// ---- POUs/Station/FB_StationTakeLoad.TcPOU
FUNCTION_BLOCK FB_StationTakeLoad
VAR_INPUT
	Enable:				BOOL;
	System:				REFERENCE TO ST_System;
	Station:			REFERENCE TO ST_SystemStation;
	Error:				REFERENCE TO ST_Error;
	Setting:			REFERENCE TO ST_Setting;
	Recipe:				REFERENCE TO ST_Recipe;	
	Parameter:			REFERENCE TO ST_StationTakeLoad;
END_VAR
VAR_OUTPUT
END_VAR
VAR
	_i:					INT;
	_arrTon:		    ARRAY[0..20] OF TON;
	_arrFbErrorTag:		ARRAY[0..20] OF FB_ErrorTag;
	_arrState:			ARRAY[0..20] OF BOOL;
	
	_iMoveAbsIndex1:	UINT;
	_iMoveAbsIndex2:	UINT;
	_bIsZWork:			BOOL;// 取Line0为真 其他情况为假
	_stHandshake: ST_StationTakeLoadHandshake;
END_VAR

A_Auto();
A_Home();

ACTION A_Auto:
CASE Station.iStepNow OF
	1000:
		Station.arrInfo[E_Language.Chinese]:="初始化完成 等待启动";
		IF Enable THEN
			Station.iStepNext:=1101;
		END_IF
	1101:
		Station.arrInfo[E_Language.Chinese]:="取料信号判断";
		Parameter.eState:=E_StationState.Load;
		Setting.eTakeModeBuffer:=E_TakeMode.None;
		Station.iStepNext:=1111;
	1111:
		IF Setting.eTakeModeBuffer=E_TakeMode.None THEN
			Setting.eTakeModeBuffer:=Setting.eTakeMode;
		ELSE
			Parameter.eState:=E_StationState.Busy;
			Station.iStepNext:=1151;
		END_IF
	1151:
		Station.arrInfo[E_Language.Chinese]:="请求取料";
		CASE Setting.eTakeModeBuffer OF
			E_TakeMode.Take0:
				_iMoveAbsIndex1:=2;
				_bIsZWork:=TRUE;
				Parameter.stHandshake.bRequestLine0Buffer_T0 :=TRUE;
				IF Parameter.stHandshake.bResponseTake_T0 THEN
					Station.iStepNext:=1201;
				END_IF
			E_TakeMode.Take1:
				_iMoveAbsIndex1:=3;
				_bIsZWork:=FALSE;
				Parameter.stHandshake.bRequestLineLoad_T1:=TRUE;
				IF Parameter.stHandshake.bResponseTake_T1 THEN
					Station.iStepNext:=1201;
				END_IF
			E_TakeMode.Take3Load:
				_iMoveAbsIndex1:=4;
				_bIsZWork:=FALSE;
				Parameter.stHandshake.bRequestLineLoad_T3:=TRUE;
				IF Parameter.stHandshake.bResponseTake_T3 THEN
					Station.iStepNext:=1201;
				END_IF
			E_TakeMode.None:
				Station.iStepNext:=1101;
		END_CASE
	1201:
		Station.arrInfo[E_Language.Chinese]:="Y轴至取料位";
		Parameter.eState:=E_StationState.Busy;
		IF Parameter.fbTakeY.M_MoveAbs(_iMoveAbsIndex1) THEN
			Station.iStepNext:=1301;
		END_IF
	1301:
		Station.arrInfo[E_Language.Chinese]:="Z模组下降";
		IF M_ZWork()  THEN
			Station.iStepNext:=1401;
		END_IF
	1401:
		Station.arrInfo[E_Language.Chinese]:="夹紧气缸夹紧";
		IF Parameter.fbTakeClamp.M_WorkRequest() THEN
			Station.iStepNext:=1501;
		END_IF
	1501:
		Station.arrInfo[E_Language.Chinese]:="Z模组上升";
		IF M_ZHome() THEN
			Station.iStepNext:=1511;
		END_IF
	1511:
		Station.arrInfo[E_Language.Chinese]:="复位取料请求 ";
		CASE Setting.eTakeModeBuffer OF
			E_TakeMode.Take0:
				Parameter.stHandshake.bRequestLine0Buffer_T0 :=FALSE;
				IF NOT Parameter.stHandshake.bResponseTake_T0 THEN
					Station.iStepNext:=1601;
				END_IF
			E_TakeMode.Take1:
				Parameter.stHandshake.bRequestLineLoad_T1:=FALSE;
				IF NOT Parameter.stHandshake.bResponseTake_T1 THEN
					Station.iStepNext:=1601;
				END_IF
			E_TakeMode.Take3Load:
				Parameter.stHandshake.bRequestLineLoad_T3:=FALSE;
				IF NOT Parameter.stHandshake.bResponseTake_T3 THEN
					Station.iStepNext:=1601;
				END_IF
		END_CASE
	1601:
		Station.arrInfo[E_Language.Chinese]:="请求放料";
		Parameter.eState:=E_StationState.Done;
		Setting.eTakeModeBuffer:=E_TakeMode.None;
		Station.iStepNext:=1611;
	1611:
		IF Setting.eTakeModeBuffer=E_TakeMode.None THEN
			Setting.eTakeModeBuffer:=Setting.eTakeMode;
		ELSE
			Parameter.eState:=E_StationState.Busy;
			Station.iStepNext:=1651;
		END_IF
	1651:
		_bIsZWork:=FALSE;
		CASE Setting.eTakeModeBuffer OF
			E_TakeMode.Place1:
				_iMoveAbsIndex2:=3;
				Parameter.stHandshake.bRequestLineLoad_P1:=TRUE;
				IF Parameter.stHandshake.bResponseTake_P1 THEN
					Station.iStepNext:=1701;
				END_IF
			E_TakeMode.Place3Load:
				_iMoveAbsIndex2:=4;
				Parameter.stHandshake.bRequestLineLoad_P3:=TRUE;
				IF Parameter.stHandshake.bResponseTake_P3 THEN
					Station.iStepNext:=1701;
				END_IF
		END_CASE
	1701:
		Station.arrInfo[E_Language.Chinese]:="等待Y轴至放料位";
		IF Parameter.fbTakeY.M_MoveAbs(_iMoveAbsIndex2) THEN
			Station.iStepNext:=1801;
		END_IF
	1801:
		Station.arrInfo[E_Language.Chinese]:="Z模组下降";
		IF M_ZWork() THEN
			Station.iStepNext:=1901;
		END_IF
	1901:
		Station.arrInfo[E_Language.Chinese]:="夹紧气缸松开";
		IF Parameter.fbTakeClamp.M_HomeRequest() THEN
			Station.iStepNext:=2001;
		END_IF
	2001:
		Station.arrInfo[E_Language.Chinese]:="Z模组上升";
		IF M_ZHome() THEN
			Station.iStepNext:=2101;
		END_IF
	2101:
		Station.arrInfo[E_Language.Chinese]:="复位放料请求";
		CASE Setting.eTakeModeBuffer OF
			E_TakeMode.Place1:
				Parameter.stHandshake.bRequestLineLoad_P1:=FALSE;
				IF NOT Parameter.stHandshake.bResponseTake_P1 THEN
					Station.iStepNext:=2201;
				END_IF
			E_TakeMode.Place3Load:
				Parameter.stHandshake.bRequestLineLoad_P3:=FALSE;
				IF NOT Parameter.stHandshake.bResponseTake_P3 THEN
					Station.iStepNext:=2201;
				END_IF
		END_CASE
	2201:
		Station.arrInfo[E_Language.Chinese]:="Y轴至初始位";
		IF Parameter.fbTakeY.M_MoveAbs(1) THEN
			Station.iStepNext:=1101;
		END_IF
END_CASE
END_ACTION

ACTION A_Home:
CASE Station.iStepNow OF
	0:
		Station.arrInfo[E_Language.Chinese]:="等待初始化";
		Parameter.stHandshake:=_stHandshake;
		Parameter.eState:=E_StationState.None;
		Setting.eTakeModeBuffer:=E_TakeMode.None;
		Station.iStepNext:=SEL(Enable,1000,500);
	500:
		Station.arrInfo[E_Language.Chinese]:="夹紧气缸松开";
		IF Parameter.fbTakeClamp.M_HomeRequest() THEN
			Station.iStepNext:=600;
		END_IF
	600:
		Station.arrInfo[E_Language.Chinese]:="Z模组初始化";
		IF M_ZInit() THEN
			Station.iStepNext:=700;
		END_IF
	700:
		Station.arrInfo[E_Language.Chinese]:="Z模组至上升位";
		IF M_ZHome() THEN
			Station.iStepNext:=800;
		END_IF
	800:
		Station.arrInfo[E_Language.Chinese]:="Y模组回零";
		IF Parameter.fbTakeY.M_Home() THEN
			Station.iStepNext:=900;
		END_IF
	900:
		Station.arrInfo[E_Language.Chinese]:="Y模组至初始位";
		IF Parameter.fbTakeY.M_MoveAbs(1) THEN
			Station.iStepNext:=1000;
		END_IF
END_CASE
END_ACTION

METHOD M_ZHome : BOOL
VAR_INPUT
END_VAR
CASE Recipe.eMachineType OF
	E_MachineType.LH311,E_MachineType.RH311:
		M_ZHome:=Parameter.fbTakeLift1.M_HomeRequest() AND Parameter.fbTakeLift2.M_HomeRequest();
	E_MachineType.LH353,E_MachineType.RH353:
		M_ZHome:=Parameter.fbTakeZ.M_MoveAbs(1);
	E_MachineType.LH367,E_MachineType.RH367:
		M_ZHome:=Parameter.fbTakeLift1.M_HomeRequest() AND Parameter.fbTakeLift2.M_HomeRequest();
	E_MachineType.LH201,E_MachineType.RH201:
		M_ZHome:=Parameter.fbTakeZ.M_MoveAbs(1);
	E_MachineType.LH069,E_MachineType.RH069:
		M_ZHome:=Parameter.fbTakeZ.M_MoveAbs(1);
	E_MachineType.LH373,E_MachineType.RH373:
		M_ZHome:=Parameter.fbTakeZ.M_MoveAbs(1);
END_CASE
END_METHOD

METHOD M_ZInit : BOOL
VAR_INPUT
END_VAR
CASE Recipe.eMachineType OF
	E_MachineType.LH311,E_MachineType.RH311:
		M_ZInit:=TRUE;
	E_MachineType.LH353,E_MachineType.RH353:
		M_ZInit:=Parameter.fbTakeZ.M_Home();
	E_MachineType.LH367,E_MachineType.RH367:
		M_ZInit:=TRUE;
	E_MachineType.LH201,E_MachineType.RH201:
		M_ZInit:=Parameter.fbTakeZ.M_Home();
	E_MachineType.LH069,E_MachineType.RH069:
		M_ZInit:=Parameter.fbTakeZ.M_Home();
	E_MachineType.LH373,E_MachineType.RH373:
		M_ZInit:=Parameter.fbTakeZ.M_Home();
END_CASE
END_METHOD

METHOD M_ZWork : BOOL
VAR_INPUT
END_VAR
CASE Recipe.eMachineType OF
	E_MachineType.LH311,E_MachineType.RH311:
		M_ZWork:=Parameter.fbTakeLift1.M_WorkRequest() AND Parameter.fbTakeLift2.M_WorkRequest();
	E_MachineType.LH353,E_MachineType.RH353:
		M_ZWork:=SEL(_bIsZWork,Parameter.fbTakeZ.M_MoveAbs(3) ,Parameter.fbTakeZ.M_MoveAbs(2));
	E_MachineType.LH367,E_MachineType.RH367:
		M_ZWork:=Parameter.fbTakeLift1.M_WorkRequest() AND SEL(_bIsZWork,TRUE ,Parameter.fbTakeLift2.M_WorkRequest()) ;
	E_MachineType.LH201,E_MachineType.RH201:
		M_ZWork:=SEL(_bIsZWork,Parameter.fbTakeZ.M_MoveAbs(3) ,Parameter.fbTakeZ.M_MoveAbs(2));
	E_MachineType.LH069,E_MachineType.RH069:
		M_ZWork:=SEL(_bIsZWork,Parameter.fbTakeZ.M_MoveAbs(3) ,Parameter.fbTakeZ.M_MoveAbs(2));
	E_MachineType.LH373,E_MachineType.RH373:
		M_ZWork:=SEL(_bIsZWork,Parameter.fbTakeZ.M_MoveAbs(3) ,Parameter.fbTakeZ.M_MoveAbs(2));
END_CASE
END_METHOD

END_FUNCTION_BLOCK

// ---- POUs/Station/FB_StationDismantling.TcPOU
FUNCTION_BLOCK FB_StationDismantling
VAR_INPUT
	Enable:				BOOL;
	System:				REFERENCE TO ST_System;
	Station:			REFERENCE TO ST_SystemStation;
	Error:				REFERENCE TO ST_Error;
	Setting:			REFERENCE TO ST_Setting;
	Recipe:				REFERENCE TO ST_Recipe;	
	Parameter:			REFERENCE TO ST_StationDismantling;	
END_VAR
VAR_OUTPUT
END_VAR
VAR
	_i:					INT;
	_arrTon:		    ARRAY[0..20] OF TON;
	_arrFbErrorTag:		ARRAY[0..20] OF FB_ErrorTag;
	_arrState:			ARRAY[0..20] OF BOOL;
	_bOpenLockTemp:		BOOL;
	_bResetLockTemp:	BOOL;
	_stHandshake:		ST_StationDismantlingHandshake;
END_VAR

A_Home();
A_Auto();

ACTION A_Auto:
CASE Station.iStepNow OF
	1000:
		Station.arrInfo[E_Language.Chinese]:="初始化完成 等待启动";
		IF  Enable THEN
			Station.iStepNext:=1101;
		END_IF
	1101:
		Station.arrInfo[E_Language.Chinese]:="判断是否有料";
		Parameter.eState:=E_StationState.Busy;
		IF NOT Parameter.bClose AND NOT Parameter.bPalletCheck2 THEN
			Station.iStepNext:=1201;
		END_IF
	1201:
		Station.arrInfo[E_Language.Chinese]:="请求放料";
		Parameter.eState:=E_StationState.Load;
		Station.iStepNext:=1301;
	1301:
		Parameter.stHandshake.bRequestLineLoad_D:=TRUE;
		IF Parameter.stHandshake.bResponseDismantling_D THEN
			Parameter.eState:=E_StationState.Busy;
			Station.iStepNext:=1401;
		END_IF
	1401:
		Station.arrInfo[E_Language.Chinese]:="等待产品流入";
		IF Parameter.bPalletCheck2 THEN
			Station.iStepNext:=1501;
		END_IF
	1501:
		Station.arrInfo[E_Language.Chinese]:="复位放料请求";
		Parameter.stHandshake.bRequestLineLoad_D:=FALSE;
		IF NOT Parameter.stHandshake.bResponseDismantling_D THEN
			Station.iStepNext:=1601;
		END_IF
	1601:
		Station.arrInfo[E_Language.Chinese]:="等待产品到位";
		IF Parameter.bPalletCheck2 THEN
			Station.iStepNext:=1701;
		END_IF
	1701:
		Station.arrInfo[E_Language.Chinese]:="顶升气缸上升 阻挡气缸缩回";
		_bOpenLockTemp:=FALSE;
		_arrState[0]:=Parameter.fbLift.M_WorkRequest() ;
		_arrState[1]:=Parameter.fbPrevent.M_HomeRequest();
		IF _arrState[0] AND _arrState[1]THEN
			Station.iStepNext:=1801;
		END_IF
	1801:
		Station.arrInfo[E_Language.Chinese]:="载具解锁";
		IF M_OpenLock() THEN
			Station.iStepNext:=1901;
		END_IF
	1901:
		Station.arrInfo[E_Language.Chinese]:="校平气缸伸出";
		IF M_StandardWork() THEN
			Station.iStepNext:=2001;
		END_IF
	2001:
		Station.arrInfo[E_Language.Chinese]:="请求取UC";
		Parameter.stHandshake.bRequestUc:=TRUE;
		IF Parameter.stHandshake.bResponseDismantling_Uc THEN
			Station.iStepNext:=2201;
		END_IF
	2201:
		Parameter.stHandshake.bRequestUc:=FALSE;
		IF NOT Parameter.stHandshake.bResponseDismantling_Uc THEN
			Station.iStepNext:=2301;
		END_IF
	2301:
		Station.arrInfo[E_Language.Chinese]:="校平气缸缩回";
		_bResetLockTemp:=FALSE;
		IF M_StandardHome() THEN
			Station.iStepNext:=2401;
		END_IF
	2401:
		Station.arrInfo[E_Language.Chinese]:="载具复位";
		IF M_ResetLock() THEN
			Station.iStepNext:=2501;
		END_IF
	2501:
		Station.arrInfo[E_Language.Chinese]:="判断下工装站是否屏蔽";
		IF NOT  Parameter.bCloseUnloadElevator THEN
			Station.iStepNext:=2551;
		ELSIF Parameter.fbLift.M_HomeRequest() THEN
			Station.iStepNext:=2801;
		END_IF
	2551:
		Station.arrInfo[E_Language.Chinese]:="请求下工装";
		Parameter.stHandshake.bRequestElevator:=TRUE;
		IF Parameter.stHandshake.bResponseDismantling_E THEN
			Station.iStepNext:=2601;
		END_IF
	2601:
		Station.arrInfo[E_Language.Chinese]:="顶升气缸下降";
		IF Parameter.fbLift.M_HomeRequest() THEN
			Station.iStepNext:=2701;
		END_IF
	2701:
		Station.arrInfo[E_Language.Chinese]:="复位请求";
		Parameter.stHandshake.bRequestElevator:=FALSE;
		IF NOT Parameter.stHandshake.bResponseDismantling_E THEN
			Station.iStepNext:=2801;
		END_IF
	2801:
		Station.arrInfo[E_Language.Chinese]:="等待产品流出";
		IF NOT Parameter.bPalletCheck1 AND NOT Parameter.bPalletCheck2 AND NOT Parameter.bPalletCheck3 THEN
			Station.iStepNext:=2901;
		END_IF
	2901:
		Station.arrInfo[E_Language.Chinese]:="阻挡气缸伸出";
		IF  Parameter.fbPrevent.M_WorkRequest() THEN
			Station.iStepNext:=1101;
		END_IF
END_CASE
END_ACTION

ACTION A_Home:
CASE Station.iStepNow OF
	0:
		Station.arrInfo[E_Language.Chinese]:="等待初始化";
		Parameter.stHandshake:=_stHandshake;
		Parameter.eState:=E_StationState.Done;
		Station.iStepNext:=SEL(Enable,1000,100);
	100:
		Station.arrInfo[E_Language.Chinese]:="阻挡气缸伸出";
		IF Parameter.fbPrevent.M_WorkRequest() THEN
			Station.iStepNext:=200;
		END_IF
	200:
		Station.arrInfo[E_Language.Chinese]:="侧推气缸缩回";
		IF M_LateralHome() THEN
			Station.iStepNext:=300;
		END_IF
	300:
		Station.arrInfo[E_Language.Chinese]:="旋转气缸复位";
		IF Parameter.fbRotate.M_HomeRequest() THEN
			Station.iStepNext:=400;
		END_IF
	400:
		Station.arrInfo[E_Language.Chinese]:="校平气缸缩回";
		IF M_StandardHome() THEN
			Station.iStepNext:=500;
		END_IF
	500:
		Station.arrInfo[E_Language.Chinese]:="顶升气缸缩回";
		IF Parameter.fbLift.M_HomeRequest() THEN
			Station.iStepNext:=1000;
		END_IF
END_CASE
END_ACTION

METHOD M_LateralHome : BOOL
VAR_INPUT
END_VAR
VAR
	_temp:			ARRAY[0..10] OF BOOL;
END_VAR
CASE Recipe.eMachineType OF
	E_MachineType.LH311,E_MachineType.RH311:
		M_LateralHome:=Parameter.fbLateral1.M_HomeRequest();
	E_MachineType.LH353,E_MachineType.RH353:
		_temp[0]:=Parameter.fbLateral1.M_HomeRequest();
		_temp[1]:=Parameter.fbLateral2.M_HomeRequest();
		M_LateralHome:=_temp[0] AND _temp[1];
	E_MachineType.LH367,E_MachineType.RH367:
		_temp[0]:=Parameter.fbLateral1.M_HomeRequest();
		_temp[1]:=Parameter.fbLateral2.M_HomeRequest();
		M_LateralHome:=_temp[0] AND _temp[1];
	E_MachineType.LH201,E_MachineType.RH201:
		_temp[0]:=Parameter.fbLateral1.M_HomeRequest();
		_temp[1]:=Parameter.fbLateral2.M_HomeRequest();
		M_LateralHome:=_temp[0] AND _temp[1];
	E_MachineType.LH069,E_MachineType.RH069:
		_temp[0]:=Parameter.fbLateral1.M_HomeRequest();
		_temp[1]:=Parameter.fbLateral2.M_HomeRequest();
		M_LateralHome:=_temp[0] AND _temp[1];
	E_MachineType.LH373,E_MachineType.RH373:
		M_LateralHome:=Parameter.fbLateral1.M_HomeRequest();
END_CASE
END_METHOD

METHOD M_LateralWork : BOOL
VAR_INPUT
END_VAR

VAR
	_temp: array[0..10] of bool;
END_VAR
CASE Recipe.eMachineType OF
	E_MachineType.LH311,E_MachineType.RH311:
		M_LateralWork:=Parameter.fbLateral1.M_WorkRequest();
	E_MachineType.LH353,E_MachineType.RH353:
		_temp[0]:=Parameter.fbLateral1.M_WorkRequest();
		_temp[1]:=Parameter.fbLateral2.M_WorkRequest();
		M_LateralWork:=_temp[0] AND _temp[1];
	E_MachineType.LH367,E_MachineType.RH367:
		_temp[0]:=Parameter.fbLateral1.M_WorkRequest();
		_temp[1]:=Parameter.fbLateral2.M_WorkRequest();
		M_LateralWork:=_temp[0] AND _temp[1];
	E_MachineType.LH201,E_MachineType.RH201:
		_temp[0]:=Parameter.fbLateral1.M_WorkRequest();
		_temp[1]:=Parameter.fbLateral2.M_WorkRequest();
		M_LateralWork:=_temp[0] AND _temp[1];
	E_MachineType.LH069,E_MachineType.RH069:
		_temp[0]:=Parameter.fbLateral1.M_WorkRequest();
		_temp[1]:=Parameter.fbLateral2.M_WorkRequest();
		M_LateralWork:=_temp[0] AND _temp[1];
	E_MachineType.LH373,E_MachineType.RH373:
		M_LateralWork:=Parameter.fbLateral1.M_WorkRequest();
END_CASE
END_METHOD

METHOD M_OpenLock : BOOL
VAR_INPUT
END_VAR
IF Recipe.eMachineType=E_MachineType.LH311 OR Recipe.eMachineType=E_MachineType.RH311 THEN
	IF M_LateralWork() THEN
		M_OpenLock:=Parameter.fbRotate.M_WorkRequest();
	END_IF
ELSE
	IF NOT _bOpenLockTemp THEN
		IF M_LateralWork() THEN
			_bOpenLockTemp:=Parameter.fbRotate.M_WorkRequest();
		END_IF
	ELSE
		CASE  Recipe.eMachineType OF
			E_MachineType.LH201,E_MachineType.RH201:
				M_OpenLock:=Parameter.fbLateral2.M_HomeRequest();
			ELSE
				M_OpenLock:=M_LateralHome();
		END_CASE
	END_IF
END_IF
END_METHOD

METHOD M_ResetLock : BOOL
VAR_INPUT
END_VAR
IF Recipe.eMachineType=E_MachineType.LH311 OR Recipe.eMachineType=E_MachineType.RH311 THEN
	IF M_LateralHome() THEN
		M_ResetLock:=Parameter.fbRotate.M_HomeRequest();;
	END_IF
ELSE
	IF NOT _bResetLockTemp THEN
		IF Parameter.fbLateral1.M_WorkRequest() THEN
			_bResetLockTemp:=Parameter.fbRotate.M_HomeRequest();
		END_IF
	ELSE
		M_ResetLock:=Parameter.fbLateral1.M_HomeRequest();
	END_IF
END_IF
END_METHOD

METHOD M_StandardHome : BOOL
VAR_INPUT
END_VAR
VAR
	_temp:			ARRAY[0..10] OF BOOL;
END_VAR
CASE Recipe.eMachineType OF
	E_MachineType.LH311,E_MachineType.RH311:
		_temp[0]:=Parameter.fbStandard1.M_HomeRequest();
		_temp[1]:=Parameter.fbStandard2.M_HomeRequest();
		M_StandardHome:=_temp[0] AND _temp[1];
	E_MachineType.LH353,E_MachineType.RH353:
		M_StandardHome:=Parameter.fbStandard1.M_HomeRequest();
	E_MachineType.LH367,E_MachineType.RH367:
		M_StandardHome:=Parameter.fbStandard1.M_HomeRequest();
	E_MachineType.LH201,E_MachineType.RH201:
		M_StandardHome:=TRUE;
	E_MachineType.LH069,E_MachineType.RH069:
		M_StandardHome:=TRUE;
	E_MachineType.LH373,E_MachineType.RH373:
		M_StandardHome:=Parameter.fbStandard1.M_HomeRequest();
END_CASE
END_METHOD

METHOD M_StandardWork : BOOL
VAR_INPUT
END_VAR

VAR
	_temp: array[0..10] of bool;
END_VAR
CASE Recipe.eMachineType OF
	E_MachineType.LH311,E_MachineType.RH311:
		_temp[0]:=Parameter.fbStandard1.M_WorkRequest();
		_temp[1]:=Parameter.fbStandard2.M_WorkRequest();
		M_StandardWork:=_temp[0] AND _temp[1];
	E_MachineType.LH353,E_MachineType.RH353:
		M_StandardWork:=Parameter.fbStandard1.M_WorkRequest();
	E_MachineType.LH367,E_MachineType.RH367:
		M_StandardWork:=Parameter.fbStandard1.M_WorkRequest();
	E_MachineType.LH201,E_MachineType.RH201:
		M_StandardWork:=TRUE;
	E_MachineType.LH069,E_MachineType.RH069:
		M_StandardWork:=TRUE;
	E_MachineType.LH373,E_MachineType.RH373:
		M_StandardWork:=TRUE;//Parameter.fbStandard1.M_WorkRequest();
END_CASE
END_METHOD

END_FUNCTION_BLOCK

// ---- POUs/Station/FB_StationLine0Load.TcPOU
FUNCTION_BLOCK FB_StationLine0Load
VAR_INPUT
	Enable:				BOOL;
	System:				REFERENCE TO ST_System;
	Station:			REFERENCE TO ST_SystemStation;
	Error:				REFERENCE TO ST_Error;
	Setting:			REFERENCE TO ST_Setting;
	Recipe:				REFERENCE TO ST_Recipe;	
	Parameter:			REFERENCE TO ST_StationLine0Load;
END_VAR
VAR_OUTPUT
END_VAR
VAR
	_i:					INT;
	_arrTon:		    ARRAY[0..20] OF TON;
	_arrFbErrorTag:		ARRAY[0..20] OF FB_ErrorTag;
	_arrState:			ARRAY[0..20] OF BOOL;
	
	_stHandshake:		ST_StationLine0LoadHandshake;
END_VAR

A_Home();
A_Auto();

ACTION A_Auto:
CASE Station.iStepNow OF
	1000:
		Station.arrInfo[E_Language.Chinese]:="初始化完成 等待启动";
		IF Enable THEN
			Station.iStepNext:=1100;
		END_IF
	1100:
		Station.arrInfo[E_Language.Chinese]:="判断阻挡位是否有料";
		IF Parameter.bPreventCheck THEN
			Station.iStepNext:=1601;
		ELSE
			Station.iStepNext:=1201;
		END_IF
	1201:
		Station.arrInfo[E_Language.Chinese]:="判断分料位是否有料";
		IF Parameter.bPartCheck AND Recipe.eLoadClose<>E_LoadClose.Line0 THEN
			Station.iStepNext:=1301;
		END_IF
	1301:
		Station.arrInfo[E_Language.Chinese]:="分料气缸缩回";
		IF  Parameter.fbPart.M_HomeRequest() THEN
			Station.iStepNext:=1401;
		END_IF
	1401:
		Station.arrInfo[E_Language.Chinese]:="等待产品至阻挡位";
		IF Parameter.bPreventCheck THEN
			Station.iStepNext:=1501;
		END_IF
	1501:
		Station.arrInfo[E_Language.Chinese]:="分料气缸伸出";
		IF  Parameter.fbPart.M_WorkRequest() THEN
			Station.iStepNext:=1601;
		END_IF
	1601:
		Station.arrInfo[E_Language.Chinese]:="等待缓存工站请求放料";
		IF Parameter.stHandshake.bRequestLine0Load THEN
			Parameter.stHandshake.bResponseLine0Buffer:=TRUE;
			Station.iStepNext:=1701;
		END_IF
	1701:
		Station.arrInfo[E_Language.Chinese]:="阻挡气缸缩回";
		IF Parameter.fbPrevent.M_HomeRequest() THEN
			Station.iStepNext:=1751;
		END_IF
	1751:
		Station.arrInfo[E_Language.Chinese]:="等待产品流出";
		IF NOT Parameter.bPreventCheck THEN
			Station.iStepNext:=1801;
		END_IF
	1801:
		Station.arrInfo[E_Language.Chinese]:="等待放料完成";
		IF NOT Parameter.stHandshake.bRequestLine0Load THEN
			Parameter.stHandshake.bResponseLine0Buffer:=FALSE;
			Station.iStepNext:=1901;
		END_IF
	1901:
		Station.arrInfo[E_Language.Chinese]:="阻挡气缸伸出";
		IF Parameter.fbPrevent.M_WorkRequest() THEN
			Station.iStepNext:=1100;
		END_IF
END_CASE
END_ACTION

ACTION A_Home:
CASE Station.iStepNow OF
	0:
		Station.arrInfo[E_Language.Chinese]:="等待初始化";
		Parameter.stHandshake:=_stHandshake;
		Station.iStepNext:=SEL(Enable,1000,200);
	200:
		Station.arrInfo[E_Language.Chinese]:="分料气缸 阻挡气缸伸出";
		_arrState[0]:=Parameter.fbPart.M_WorkRequest();
		_arrState[1]:=Parameter.fbPrevent.M_WorkRequest();
		IF _arrState[0] AND _arrState[1] THEN
			Station.iStepNext:=1000;
		END_IF
END_CASE
END_ACTION

END_FUNCTION_BLOCK

// ---- POUs/Station/FB_StationLine0Buffer.TcPOU
FUNCTION_BLOCK FB_StationLine0Buffer
VAR_INPUT
	Enable:				BOOL;
	System:				REFERENCE TO ST_System;
	Station:			REFERENCE TO ST_SystemStation;
	Error:				REFERENCE TO ST_Error;
	Setting:			REFERENCE TO ST_Setting;
	Recipe:				REFERENCE TO ST_Recipe;	
	Parameter:			REFERENCE TO ST_StationLine0Buffer;	
END_VAR
VAR_OUTPUT
END_VAR
VAR
	_i:					INT;
	_arrTon:		    ARRAY[0..20] OF TON;
	_arrFbErrorTag:		ARRAY[0..20] OF FB_ErrorTag;
	_arrState:			ARRAY[0..20] OF BOOL;
	
	_stHandshake:		ST_StationLine0BufferHandshake;
END_VAR

A_Home();
A_Auto();

ACTION A_Auto:
CASE Station.iStepNow OF
	1000:
		Station.arrInfo[E_Language.Chinese]:="初始化完成 等待启动";
		IF Enable THEN
			Station.iStepNext:=1101;
		END_IF
	1101:
		Station.arrInfo[E_Language.Chinese]:="判断缓存位是否有料";
		Parameter.eState:=E_StationState.Busy;
		IF Parameter.bPlace AND NOT GVL.stSetting.bDryRun THEN
			Station.iStepNext:=1501;
		ELSE
			Station.iStepNext:=1201;
		END_IF
	1201:
		Station.arrInfo[E_Language.Chinese]:="请求上料站放料";
		Parameter.stHandshake.bRequestLine0Load:=TRUE;
		IF Parameter.stHandshake.bResponseLine0Buffer THEN
			Station.iStepNext:=1301;
		END_IF
	1301:
		Station.arrInfo[E_Language.Chinese]:="等待产品到位";
		IF Parameter.bPlace THEN
			Station.iStepNext:=1401;
		END_IF
	1401:
		Station.arrInfo[E_Language.Chinese]:="复位请求信号";
		Parameter.stHandshake.bRequestLine0Load:=FALSE;
		IF NOT Parameter.stHandshake.bResponseLine0Buffer THEN
			Station.iStepNext:=1501;
		END_IF
	1501:
		Station.arrInfo[E_Language.Chinese]:="取料信号判断";
		Parameter.eState:=E_StationState.Done;
		Station.iStepNext:=1511;
	1511:
		IF Setting.eTakeModeBuffer=E_TakeMode.Take0 THEN
			Parameter.eState:=E_StationState.Busy;
			Station.iStepNext:=1551;
		END_IF
	1551:
		Station.arrInfo[E_Language.Chinese]:="等取料站取料请求";
		IF Parameter.stHandshake.bRequestLine0Buffer_T THEN
			Parameter.stHandshake.bResponseTake_T:=TRUE;
			Station.iStepNext:=1601;
		END_IF
	1601:
		Station.arrInfo[E_Language.Chinese]:="等待取料站取料完成";
		IF NOT Parameter.stHandshake.bRequestLine0Buffer_T THEN
			Parameter.stHandshake.bResponseTake_T:=FALSE;
			Station.iStepNext:=1101;
		END_IF
END_CASE
END_ACTION

ACTION A_Home:
CASE Station.iStepNow OF
	0:
		Station.arrInfo[E_Language.Chinese]:="等待初始化";
		Parameter.eState:=E_StationState.None;
		Parameter.stHandshake:=_stHandshake;
		Station.iStepNext:=1000;
END_CASE
END_ACTION

END_FUNCTION_BLOCK

// ---- POUs/Station/FB_StationLineLoad.TcPOU
FUNCTION_BLOCK FB_StationLineLoad
VAR_INPUT
	Enable:				BOOL;
	System:				REFERENCE TO ST_System;
	Station:			REFERENCE TO ST_SystemStation;
	Error:				REFERENCE TO ST_Error;
	Setting:			REFERENCE TO ST_Setting;
	Recipe:				REFERENCE TO ST_Recipe;
	Parameter:			REFERENCE TO ST_StationLineLoad;
END_VAR
VAR_OUTPUT
END_VAR
VAR
	_i:					INT;
	_arrTon:		    ARRAY[0..20] OF TON;
	_arrFbErrorTag:		ARRAY[0..20] OF FB_ErrorTag;
	_arrState:			ARRAY[0..20] OF BOOL;
	
	_stHandshake:		ST_StationLineLoadHandshake;
END_VAR

A_Home();
A_Auto();

_arrTon[0](IN:=System.stInput.bStart , PT:=T#3S , Q=> , ET=> );

ACTION A_Auto:
CASE Station.iStepNow OF
	1000:
		Station.arrInfo[E_Language.Chinese]:="初始化完成 等待启动";
		IF Enable THEN
			Station.iStepNext:=1101;
		END_IF
	1101:
		Station.arrInfo[E_Language.Chinese]:="判断线体是否关闭";
		Parameter.eState:=E_StationState.Busy;
		 IF NOT Parameter.bIsClosed THEN
			 Station.iStepNext:=SEL(Parameter.bManualLoad,1201,1151);
		 END_IF
	1151:
		Station.arrInfo[E_Language.Chinese]:="等待手动上料后启动";
		IF _arrTon[0].Q THEN
			Station.iStepNext:=1701;
		END_IF
	1201:
		Station.arrInfo[E_Language.Chinese]:="请求放料";
		Parameter.eState:=E_StationState.Load;
		Station.iStepNext:=1211;
	1211:
		Station.arrInfo[E_Language.Chinese]:="等待上料";
		IF Parameter.stHandshake.bRequestLineLoad_P AND Station.iStepNext=Station.iStepNow THEN
			Parameter.eState:=E_StationState.Busy;
			Parameter.stHandshake.bResponseTake_P:=TRUE;
			Station.iStepNext:=1251;
		END_IF
		IF Parameter.stHandshake.bRequestTake_P_M AND NOT System.stMode.bPause AND Station.iStepNext=Station.iStepNow THEN
			Parameter.eState:=E_StationState.Busy;
			Parameter.stHandshake.bResponseMachine_P:=TRUE;
			Station.iStepNext:=1301;
		END_IF
	1251:
		Station.arrInfo[E_Language.Chinese]:="等待复位放料请求信号";
		IF NOT Parameter.stHandshake.bRequestLineLoad_P THEN
			Parameter.stHandshake.bResponseTake_P:=FALSE;
			Station.iStepNext:=1701;
		END_IF
	1301:
		Station.arrInfo[E_Language.Chinese]:="顶升及提升气缸缩回";
		_arrState[0]:=Parameter.fbLift.M_HomeRequest();
		_arrState[1]:=Parameter.fbElevator.M_HomeRequest();
		IF _arrState[0] AND _arrState[1]THEN
			Station.iStepNext:=1351;
		END_IF
	1351:
		Station.arrInfo[E_Language.Chinese]:="等待产品流入";
		IF Parameter.bPalletCheck1 THEN
			Station.iStepNext:=SEL(Parameter.bManualLoad,1401,1501);
		END_IF
	1401:
		Station.arrInfo[E_Language.Chinese]:="等待上台设备复位放料信号";
		IF NOT Parameter.stHandshake.bRequestTake_P_M  THEN
			Parameter.stHandshake.bResponseMachine_P:=FALSE;
		    Station.iStepNext:=1501;
		END_IF
	1501:
		Station.arrInfo[E_Language.Chinese]:="等待产品到位";
		IF Parameter.bPalletCheck2 THEN
			Station.iStepNext:=1601;
		END_IF
	1601:
		Station.arrInfo[E_Language.Chinese]:="顶升气缸伸出 提升气缸伸出";
		IF  Parameter.fbLift.M_WorkRequest() AND Parameter.fbElevator.M_WorkRequest() THEN
			Station.iStepNext:=1701;
		END_IF
	1701:
		Station.arrInfo[E_Language.Chinese]:="阻挡气缸缩回 调宽气缸调宽";
		_arrState[1]:=Parameter.fbPrevent.M_HomeRequest();
		_arrState[2]:=M_AdjustWork();
		IF  _arrState[1] AND _arrState[2] THEN
			Station.iStepNext:=1801;
		END_IF
	1801:
		Station.arrInfo[E_Language.Chinese]:="请求取料";
		Parameter.eState:=E_StationState.Done;
		Station.iStepNext:=1811;
	1811:
		Station.arrInfo[E_Language.Chinese]:="等待取料";
		IF Parameter.stHandshake.bRequestLineLoad_T AND Station.iStepNext=Station.iStepNow THEN
			Parameter.eState:=E_StationState.Busy;
			Parameter.stHandshake.bResponseTake_T:=TRUE;
			Station.iStepNext:=1861;
		END_IF
		IF Parameter.stHandshake.bRequestLineLoad_D AND Station.iStepNext=Station.iStepNow THEN
			Parameter.eState:=E_StationState.Busy;
			Parameter.stHandshake.bResponseDismantling_D:=TRUE;
			Station.iStepNext:=2201;
		END_IF
	1861:
		IF NOT Parameter.stHandshake.bRequestLineLoad_T THEN
			Parameter.stHandshake.bResponseTake_T:=FALSE;
			Station.iStepNext:=2501;
		END_IF
	2201:
		Station.arrInfo[E_Language.Chinese]:="旋转气缸至工作位";
		IF Parameter.fbRotate.M_WorkRequest() THEN
			Station.iStepNext:=2301;
		END_IF
	2301:
		Station.arrInfo[E_Language.Chinese]:="顶升气缸下降"; 
		IF  Parameter.fbLift.M_HomeRequest() THEN
			Station.iStepNext:=2401;
		END_IF
	2401:
		Station.arrInfo[E_Language.Chinese]:="等待产品流走";
		IF NOT Parameter.bPalletCheck2 AND NOT Parameter.bPalletCheck3 THEN
			Station.iStepNext:=2451;
		END_IF
	2451:
		Station.arrInfo[E_Language.Chinese]:="等待复位请求信号";
		IF NOT Parameter.stHandshake.bRequestLineLoad_D THEN
			Parameter.stHandshake.bResponseDismantling_D:=FALSE;
			Station.iStepNext:=2501;
		END_IF
	2501:
		Station.arrInfo[E_Language.Chinese]:="阻挡气缸伸出 调宽气缸复位 顶升气缸顶升";
		_arrState[1]:=Parameter.fbPrevent.M_WorkRequest();
		_arrState[2]:=M_AdjustHome();
		_arrState[3]:=Parameter.fbLift.M_WorkRequest();
		IF  _arrState[1] AND _arrState[2] AND _arrState[3] THEN
			Station.iStepNext:=2601;
		END_IF
	2601:
		Station.arrInfo[E_Language.Chinese]:="旋转气缸复位";
		IF Parameter.fbRotate.M_HomeRequest() THEN
			Station.iStepNext:=1101;
		END_IF
END_CASE
END_ACTION

ACTION A_Home:
CASE Station.iStepNow OF
	0:
		Station.arrInfo[E_Language.Chinese]:="等待初始化";
		Parameter.eState:=E_StationState.None;
		Parameter.stHandshake:=_stHandshake;
		Station.iStepNext:=SEL(Enable,1000,50);
	50:
		Station.arrInfo[E_Language.Chinese]:="阻挡气缸伸出";
		IF Parameter.fbPrevent.M_WorkRequest() THEN
			Station.iStepNext:=100;
		END_IF
	100:
		Station.arrInfo[E_Language.Chinese]:="提升气缸伸出";
		IF Parameter.fbElevator.M_WorkRequest() THEN
			Station.iStepNext:=200;
		END_IF
	200:
		Station.arrInfo[E_Language.Chinese]:="顶升气缸伸出";
		IF Parameter.fbLift.M_WorkRequest() THEN
			Station.iStepNext:=300;
		END_IF
	300:
		Station.arrInfo[E_Language.Chinese]:="旋转气缸复位";
		IF Parameter.fbRotate.M_HomeRequest() THEN
			Station.iStepNext:=400;
		END_IF
	400:
		Station.arrInfo[E_Language.Chinese]:="调宽气缸缩回";
		IF M_AdjustHome() THEN
			Station.iStepNext:=1000;
		END_IF
END_CASE
END_ACTION

METHOD M_AdjustHome : BOOL
VAR_INPUT
END_VAR
CASE Recipe.eMachineType OF
	E_MachineType.LH311,E_MachineType.RH311:
		M_AdjustHome:=TRUE;
	E_MachineType.LH353,E_MachineType.RH353:
		M_AdjustHome:=Parameter.fbAdjust1.M_HomeRequest();
	E_MachineType.LH367,E_MachineType.RH367:
		M_AdjustHome:=TRUE;
	E_MachineType.LH201,E_MachineType.RH201:
		M_AdjustHome:=TRUE;
	E_MachineType.LH069,E_MachineType.RH069:
		M_AdjustHome:=TRUE;
	E_MachineType.LH373,E_MachineType.RH373:
		M_AdjustHome:=Parameter.fbAdjust1.M_HomeRequest();
END_CASE
END_METHOD

METHOD M_AdjustWork : BOOL
VAR_INPUT
END_VAR
CASE Recipe.eMachineType OF
	E_MachineType.LH311,E_MachineType.RH311:
		M_AdjustWork:=TRUE;
	E_MachineType.LH353,E_MachineType.RH353:
		M_AdjustWork:=Parameter.fbAdjust1.M_WorkRequest();
	E_MachineType.LH367,E_MachineType.RH367:
		M_AdjustWork:=TRUE;
	E_MachineType.LH201,E_MachineType.RH201:
		M_AdjustWork:=TRUE;
	E_MachineType.LH069,E_MachineType.RH069:
		M_AdjustWork:=TRUE;
	E_MachineType.LH373,E_MachineType.RH373:
		M_AdjustWork:=Parameter.fbAdjust1.M_WorkRequest();
END_CASE
END_METHOD

END_FUNCTION_BLOCK

// ---- POUs/Station/FB_StationUnloadUc.TcPOU
FUNCTION_BLOCK FB_StationUnloadUc
VAR_INPUT
	Enable:				BOOL;
	System:				REFERENCE TO ST_System;
	Station:			REFERENCE TO ST_SystemStation;
	Error:				REFERENCE TO ST_Error;
	Setting:			REFERENCE TO ST_Setting;
	Recipe:				REFERENCE TO ST_Recipe;	
	Parameter:			REFERENCE TO ST_StationUnloadUc;
END_VAR
VAR_OUTPUT
END_VAR
VAR
	_i:					INT;
	_arrTon:		    ARRAY[0..20] OF TON;
	_arrFbErrorTag:		ARRAY[0..20] OF FB_ErrorTag;
	_arrState:			ARRAY[0..20] OF BOOL;
	_stHandshake: 		ST_StationUnloadUcHandshake;
END_VAR

A_Auto();
A_Home();

ACTION A_Auto:
CASE Station.iStepNow OF
	1000:
		Station.arrInfo[E_Language.Chinese]:="初始化完成 等待启动";
		IF Enable THEN
			Station.iStepNext:=1101;
		END_IF
	1101:
		Station.arrInfo[E_Language.Chinese]:="等待拆解站请求取料";
		IF Parameter.stHandshake.bRequestUc THEN
			Parameter.stHandshake.bResponseDismantling_Uc:=TRUE;
			Station.iStepNext:=1201;
		END_IF
	1201:
		Station.arrInfo[E_Language.Chinese]:="旋转气缸至取料位";
		IF Parameter.fbRotate.M_HomeRequest() THEN
			Station.iStepNext:=1251;
		END_IF
	1251:
		Station.arrInfo[E_Language.Chinese]:="升降气缸下降";
		IF  Parameter.fbLift.M_HomeRequest() THEN
			Station.iStepNext:=1301;
		END_IF
	1301:
		Station.arrInfo[E_Language.Chinese]:="夹紧气缸夹紧";
		IF Parameter.fbClamp.M_WorkRequest() THEN
			Station.iStepNext:=1401;
		END_IF
	1401:
		Station.arrInfo[E_Language.Chinese]:="升降气缸上升";
		IF Parameter.fbLift.M_WorkRequest() THEN
			Station.iStepNext:=1451;
		END_IF
	1451:
		Station.arrInfo[E_Language.Chinese]:="向下线体 请求放料";
		Parameter.stHandshake.bRequestUnloadLine:=TRUE;
		IF Parameter.stHandshake.bResponseUnladLine THEN
			Station.iStepNext:=1501;
		END_IF
	1501:
		Station.arrInfo[E_Language.Chinese]:="旋转气缸动作";
		IF Parameter.fbRotate.M_WorkRequest() THEN
			Station.iStepNext:=1551;
		END_IF
	1551:
		Station.arrInfo[E_Language.Chinese]:="等待复位取料请求";
		IF NOT Parameter.stHandshake.bRequestUc THEN
			Parameter.stHandshake.bResponseDismantling_Uc:=FALSE;
			Station.iStepNext:=1601;
		END_IF
	1601:
		Station.arrInfo[E_Language.Chinese]:="夹紧气缸松开";
		IF Parameter.fbClamp.M_HomeRequest() THEN
			Station.iStepNext:=1801;
		END_IF
	1801:
		Station.arrInfo[E_Language.Chinese]:="复位放料请求";
		Parameter.stHandshake.bRequestUnloadLine:=FALSE;
		IF NOT Parameter.stHandshake.bResponseUnladLine THEN
			Station.iStepNext:=1101;
		END_IF
END_CASE
END_ACTION

ACTION A_Home:
CASE Station.iStepNow OF
	0:
		Station.arrInfo[E_Language.Chinese]:="等待初始化";
		Parameter.stHandshake:=_stHandshake;
		Station.iStepNext:=SEL(Enable,1000,200);
	200:
		Station.arrInfo[E_Language.Chinese]:="升降气缸上升";
		IF Parameter.fbLift.M_WorkRequest() THEN
			Station.iStepNext:=300;
		END_IF
	300:
		Station.arrInfo[E_Language.Chinese]:="旋转气缸至下UC位";
		IF Parameter.fbRotate.M_WorkRequest() THEN
			Station.iStepNext:=400;
		END_IF
	400:
		Station.arrInfo[E_Language.Chinese]:="夹紧气缸复位";
		IF  Parameter.fbClamp.M_HomeRequest() THEN
			Station.iStepNext:=1000;
		END_IF
END_CASE
END_ACTION

END_FUNCTION_BLOCK

// ---- POUs/Station/FB_StationUnloadElevator.TcPOU
FUNCTION_BLOCK FB_StationUnloadElevator
VAR_INPUT
	Enable:				BOOL;
	System:				REFERENCE TO ST_System;
	Station:			REFERENCE TO ST_SystemStation;
	Error:				REFERENCE TO ST_Error;
	Setting:			REFERENCE TO ST_Setting;
	Recipe:				REFERENCE TO ST_Recipe;	
	Parameter:			REFERENCE TO ST_StationUnloadElevator;
END_VAR
VAR_OUTPUT
END_VAR
VAR
	_stHandshake: ST_StationUnloadElevatorHandshake;
END_VAR

A_Auto();
A_Home();

ACTION A_Auto:
CASE Station.iStepNow OF
	1000:
		Station.arrInfo[E_Language.Chinese]:="初始化完成 等待启动";
		IF Enable THEN
			Station.iStepNext:=1101;
		END_IF
	1101:
		Station.arrInfo[E_Language.Chinese]:="判断是否有料";
		IF NOT Parameter.bFrockElevator1NoneCheck THEN
			Station.iStepNext:=1201;
		END_IF
	1201:
		Station.arrInfo[E_Language.Chinese]:="等待拆解站请求放料";
		IF Parameter.stHandshake.bRequestElevator THEN
			Parameter.stHandshake.bResponseDismantling_E:=TRUE;
			Station.iStepNext:=1301;
		END_IF
	1301:
		Station.arrInfo[E_Language.Chinese]:="等待产品到位";
		IF Parameter.bFrockElevator1NoneCheck THEN
			Station.iStepNext:=1351;
		END_IF
	1351:
		Station.arrInfo[E_Language.Chinese]:="等待复位放料请求";
		IF NOT Parameter.stHandshake.bRequestElevator THEN
			Parameter.stHandshake.bResponseDismantling_E:=FALSE;
			Station.iStepNext:=1401;
		END_IF
	1401:
		Station.arrInfo[E_Language.Chinese]:="锁紧工装";
		IF Parameter.fbFrockRotateDown.M_HomeRequest() THEN
			Station.iStepNext:=1501;
		END_IF
	1501:
		Station.arrInfo[E_Language.Chinese]:="提升气缸上升";
		IF Parameter.fbFrockElevator.M_WorkRequest() THEN
			Station.iStepNext:=1601;
		END_IF
	1601:
		Station.arrInfo[E_Language.Chinese]:="松开工装";
		IF Parameter.fbFrockRotateDown.M_WorkRequest() THEN
			Station.iStepNext:= SEL(Parameter.bManualUnload,1701,1801);
		END_IF
	1701:
		Station.arrInfo[E_Language.Chinese]:="向下线体请求放料";
		Parameter.stHandshake.bRequestUnline:=TRUE;
		IF Parameter.stHandshake.bResponseElevator THEN
			Station.iStepNext:=1801;
		END_IF
	1801:
		Station.arrInfo[E_Language.Chinese]:="拨料气缸伸出";
		IF Parameter.fbFrockPush.M_WorkRequest() THEN
			Station.iStepNext:=1901;
		END_IF
	1901:
		Station.arrInfo[E_Language.Chinese]:="拨料气缸缩回";
		IF Parameter.fbFrockPush.M_HomeRequest() THEN
			Station.iStepNext:=SEL(Parameter.bManualUnload,2001,2101);
		END_IF
	2001:
		Station.arrInfo[E_Language.Chinese]:="复位放料请求";
		Parameter.stHandshake.bRequestUnline:=FALSE;
		IF NOT Parameter.stHandshake.bResponseElevator THEN
			Station.iStepNext:=2101;
		END_IF
	2101:
		Station.arrInfo[E_Language.Chinese]:="旋转压紧气缸缩回";
		IF Parameter.fbFrockRotateDown.M_HomeRequest() THEN
			Station.iStepNext:=2201;
		END_IF
	2201:
		Station.arrInfo[E_Language.Chinese]:="提升气缸下降";
		IF Parameter.fbFrockElevator.M_HomeRequest() THEN
			Station.iStepNext:=2301;
		END_IF
	2301:
		Station.arrInfo[E_Language.Chinese]:="旋转压紧气缸伸出";
		IF Parameter.fbFrockRotateDown.M_WorkRequest() THEN
			Station.iStepNext:=1101;
		END_IF
END_CASE
END_ACTION

ACTION A_Home:
CASE Station.iStepNow OF
	0:
		Station.arrInfo[E_Language.Chinese]:="等待初始化";
		Parameter.stHandshake:=_stHandshake;
		Station.iStepNext:=SEL(Enable,1000,100);
	100:
		Station.arrInfo[E_Language.Chinese]:="拨料气缸复位";
		IF Parameter.fbFrockPush.M_HomeRequest() THEN
			Station.iStepNext:=200;
		END_IF
	200:
		Station.arrInfo[E_Language.Chinese]:="旋转压紧气缸缩回";
		IF Parameter.fbFrockRotateDown.M_HomeRequest() THEN
			Station.iStepNext:=300;
		END_IF
	300:
		Station.arrInfo[E_Language.Chinese]:="提升气缸下降";
		IF Parameter.fbFrockElevator.M_HomeRequest() THEN
			Station.iStepNext:=400;
		END_IF
	400:
		Station.arrInfo[E_Language.Chinese]:="旋转压紧气缸伸出";
		IF Parameter.fbFrockRotateDown.M_WorkRequest() THEN
			Station.iStepNext:=1000;
		END_IF
END_CASE
END_ACTION

END_FUNCTION_BLOCK

// ---- POUs/Station/FB_StationUnloadLine.TcPOU
FUNCTION_BLOCK FB_StationUnloadLine
VAR_INPUT
	Enable:				BOOL;
	System:				REFERENCE TO ST_System;
	Station:			REFERENCE TO ST_SystemStation;
	Error:				REFERENCE TO ST_Error;
	Setting:			REFERENCE TO ST_Setting;
	Recipe:				REFERENCE TO ST_Recipe;	
	Parameter:			REFERENCE TO ST_StationUnloadLine;
END_VAR
VAR_OUTPUT
END_VAR
VAR
	_iState:			INT;// 放料请求状态
	_stHandshake: ST_StationUnloadLineHandshake;
END_VAR

A_Auto();
A_Home();

ACTION A_Auto:
CASE Station.iStepNow OF
	1000:
		Station.arrInfo[E_Language.Chinese]:="初始化完成 等待启动";
		IF Enable THEN
			Station.iStepNext:=1101;
		END_IF
	1101:
		Station.arrInfo[E_Language.Chinese]:="判断推料位是否有料";
		IF Parameter.bBeltDone AND NOT GVL.stSetting.bDryRun THEN
			Station.iStepNext:=1901;
		ELSE
			Station.iStepNext:=1201;
		END_IF
	1201:
		Station.arrInfo[E_Language.Chinese]:="判断缓存位是否有料";
		IF Parameter.bCheck1 OR Parameter.bCheck2  THEN
			Station.iStepNext:=1601;
		ELSE
			Station.iStepNext:=1301;
		END_IF
	1301:
		Station.arrInfo[E_Language.Chinese]:="等待请求放料";
		IF Parameter.stHandshake.bRequestUnloadLine2 AND Station.iStepNext=Station.iStepNow THEN
			_iState:=2;
			Parameter.stHandshake.bResponseUnladLine2:=TRUE;
			Station.iStepNext:=1601;
		END_IF
		IF Parameter.stHandshake.bRequestUnloadLine3 AND Station.iStepNext=Station.iStepNow THEN
			_iState:=3;
			Parameter.stHandshake.bResponseUnladLine3:=TRUE;
			Station.iStepNext:=1601;
		END_IF
	1601:
		Station.arrInfo[E_Language.Chinese]:="线体正转 等待到位";
		IF Parameter.fbLineAxis.M_Jog(1) AND Parameter.bBeltDone THEN
			Station.iStepNext:=1701;
		END_IF
	1701:
		Station.arrInfo[E_Language.Chinese]:="线体停止";
		IF Parameter.fbLineAxis.M_Jog(0) THEN
			Station.iStepNext:=1751;
		END_IF
	1751:
		Station.arrInfo[E_Language.Chinese]:="等待复位放料请求"; 
		CASE _iState OF
			2:// 线体2请求放料
				IF NOT Parameter.stHandshake.bRequestUnloadLine2 THEN
					Parameter.stHandshake.bResponseUnladLine2:=FALSE;
					_iState:=0;
				END_IF
			3:// 线体3请求放料
				IF NOT Parameter.stHandshake.bRequestUnloadLine3 THEN
					Parameter.stHandshake.bResponseUnladLine3:=FALSE;
					_iState:=0;
				END_IF
			ELSE
				Station.iStepNext:=1801;
		END_CASE
	1801:
		Station.arrInfo[E_Language.Chinese]:="判断下料斜坡是否有料";
		IF NOT Parameter.bBeltNoneCheck THEN
			Station.iStepNext:=SEL(Parameter.bManualUnload,1901,1851);
		END_IF
	1851:
		Station.arrInfo[E_Language.Chinese]:="等待取料";
		IF NOT Parameter.bBeltDone THEN
			Station.iStepNext:=1101;
		END_IF
	1901:
		Station.arrInfo[E_Language.Chinese]:="推料气缸伸出";
		IF Parameter.fbDrive.M_WorkRequest() THEN
			Station.iStepNext:=2001;
		END_IF
	2001:
		Station.arrInfo[E_Language.Chinese]:="推料气缸缩回";
		IF Parameter.fbDrive.M_HomeRequest() THEN
			Station.iStepNext:=1101;
		END_IF
END_CASE
END_ACTION

ACTION A_Home:
CASE Station.iStepNow OF
	0:
		Station.arrInfo[E_Language.Chinese]:="等待初始化";
		Parameter.stHandshake:=_stHandshake;
		_iState:=0;
		Station.iStepNext:=SEL(Enable,1000,100);
	100:
		Station.arrInfo[E_Language.Chinese]:="推料气缸复位";
		IF  Parameter.fbDrive.M_HomeRequest() THEN
			Station.iStepNext:=1000;
		END_IF
END_CASe
END_ACTION

END_FUNCTION_BLOCK

// ---- POUs/Station/FB_StationUnLoadUc_311.TcPOU
FUNCTION_BLOCK FB_StationUnLoadUc_311
VAR_INPUT
	Enable:				BOOL;
	System:				REFERENCE TO ST_System;
	Station:			REFERENCE TO ST_SystemStation;
	Error:				REFERENCE TO ST_Error;
	Setting:			REFERENCE TO ST_Setting;
	Recipe:				REFERENCE TO ST_Recipe;	
	Parameter:			REFERENCE TO ST_StationUnloadUc_311;
END_VAR
VAR_OUTPUT
END_VAR
VAR
	_i:					INT;
	_arrTon:		    ARRAY[0..20] OF TON;
	_arrFbErrorTag:		ARRAY[0..20] OF FB_ErrorTag;
	_arrState:			ARRAY[0..20] OF BOOL;
	_iTakeTemp:			UINT;// 取料位
	_stHandshake: ST_StationUnloadUc_311Handshake;
END_VAR

A_Home();
A_Auto();

ACTION A_Auto:
CASE Station.iStepNow OF
	1000:
		Station.arrInfo[E_Language.Chinese]:="初始化完成 等待启动";
		IF Enable THEN
			Station.iStepNext:=1101;
		END_IF
	1101:
		Station.arrInfo[E_Language.Chinese]:="等待请求取料";
		_iTakeTemp:=0;
		IF Parameter.stHandshake.bRequestUc_L2 THEN
			_iTakeTemp:=2;
		END_IF
		IF Parameter.stHandshake.bRequestUc_L3 THEN
			_iTakeTemp:=3;
		END_IF
		IF _iTakeTemp<>0 THEN
			Station.iStepNext:=1201;
		END_IF
	1201:
		CASE _iTakeTemp OF
			2:
				IF Parameter.stHandshake.bRequestUc_L2 THEN
					Parameter.stHandshake.bResponseDismantling_Uc_L2:=TRUE;
					Station.iStepNext:=1301;
				END_IF
			3:	
				IF Parameter.stHandshake.bRequestUc_L3 THEN
					Parameter.stHandshake.bResponseDismantling_Uc_L3:=TRUE;
					Station.iStepNext:=1301;
				END_IF
		END_CASE
	1301:
		Station.arrInfo[E_Language.Chinese]:="定位至取料位";
		IF Parameter.fbAxisY.M_MoveAbs(_iTakeTemp) THEN
			Station.iStepNext:=1401;
		END_IF
	1401:
		Station.arrInfo[E_Language.Chinese]:="Z气缸下降";
		IF Parameter.fbLift.M_WorkRequest() THEN
			Station.iStepNext:=1501;
		END_IF
	1501:
		Station.arrInfo[E_Language.Chinese]:="夹紧气缸夹紧";
		IF Parameter.fbClamp.M_WorkRequest() THEN
			Station.iStepNext:=1601;
		END_IF
	1601:
		Station.arrInfo[E_Language.Chinese]:="Z气缸上升";
		IF Parameter.fbLift.M_HomeRequest() THEN
			Station.iStepNext:=1651;
		END_IF
	1651:
		Station.arrInfo[E_Language.Chinese]:="等待复位请求信号";
		CASE _iTakeTemp OF
			2:
				IF NOT Parameter.stHandshake.bRequestUc_L2 THEN
					Parameter.stHandshake.bResponseDismantling_Uc_L2:=FALSE;
					Station.iStepNext:=1901;
				END_IF
			3:	
				IF NOT Parameter.stHandshake.bRequestUc_L3 THEN
					Parameter.stHandshake.bResponseDismantling_Uc_L3:=FALSE;
					Station.iStepNext:=1901;
				END_IF
		END_CASE
	1901:
		Station.arrInfo[E_Language.Chinese]:="至下UC位";
		IF Parameter.fbAxisY.M_MoveAbs(4) THEN
			Station.iStepNext:=2001;
		END_IF
	2001:
		Station.arrInfo[E_Language.Chinese]:="Z气缸 摆动下降";
		IF Parameter.fbLift.M_WorkRequest() AND Parameter.fbSwing.M_WorkRequest() THEN
			Station.iStepNext:=2101;
		END_IF
	2101:
		Station.arrInfo[E_Language.Chinese]:="夹紧气缸松开";
		IF Parameter.fbClamp.M_HomeRequest() THEN
			Station.iStepNext:=2201;
		END_IF
	2201:
		Station.arrInfo[E_Language.Chinese]:="Z气缸 摆动上升";
		IF Parameter.fbLift.M_HomeRequest() AND Parameter.fbSwing.M_HomeRequest() THEN
			Station.iStepNext:=2301;
		END_IF
	2301:
		Station.arrInfo[E_Language.Chinese]:="至初始位";
		IF Parameter.fbAxisY.M_MoveAbs(1) THEN
			Station.iStepNext:=1101;
		END_IF
END_CASE
END_ACTION

ACTION A_Home:
CASE Station.iStepNow OF
	0:
		Station.arrInfo[E_Language.Chinese]:="等待初始化";
		Parameter.stHandshake:=_stHandshake;
		Station.iStepNext:=SEL(Enable,1000,100);
	100:
		Station.arrInfo[E_Language.Chinese]:="夹紧气缸松开";
		IF Parameter.fbClamp.M_HomeRequest() THEN
			Station.iStepNext:=200;
		END_IF
	200:
		Station.arrInfo[E_Language.Chinese]:="Z气缸上升";
		IF Parameter.fbLift.M_HomeRequest() THEN
			Station.iStepNext:=250;
		END_IF
	250:
		Station.arrInfo[E_Language.Chinese]:="摆动气缸上升";
		IF Parameter.fbSwing.M_HomeRequest() THEN
			Station.iStepNext:=300;
		END_IF
	300:
		Station.arrInfo[E_Language.Chinese]:="Y轴回零";
		IF  Parameter.fbAxisY.M_Home() THEN
			Station.iStepNext:=400;
		END_IF
	400:
		Station.arrInfo[E_Language.Chinese]:="Y轴至初始位";
		IF  Parameter.fbAxisY.M_MoveAbs(1) THEN
			Station.iStepNext:=1000;
		END_IF
END_CASE
END_ACTION

END_FUNCTION_BLOCK

// ---- POUs/Device/FB_LineAxis.TcPOU
FUNCTION_BLOCK FB_LineAxis
VAR_INPUT
	System:					REFERENCE TO ST_System;
END_VAR
VAR_OUTPUT
	Moving:					BOOL;
END_VAR
VAR
	_moving:				BOOL;
END_VAR

Moving:=FALSE;

IF System.stInput.bReset THEN
	Moving:=_moving:=FALSE;
END_IF


IF System.stMode.stDeviceEnable.bAuto OR System.stMode.stDeviceEnable.bManual THEN
	Moving:=_moving;
END_IF

METHOD M_Jog : BOOL
VAR_INPUT
	Command:				INT;// -1:反转 0:停止 1:正转
END_VAR
M_Jog:=FALSE;
IF Command=1 THEN
	_moving:=TRUE;
	M_Jog:=TRUE;
END_IF

IF Command=0 THEN
	_moving:=FALSE;
	M_Jog:=TRUE;
END_IF
END_METHOD

END_FUNCTION_BLOCK

// ---- GlobalTextList.TcGTLO
TEXTLIST GlobalTextList
  109 = '  MachineType:%s'
  799 = '%dms'
  938 = 'Admin'
  145 = 'Dismantling'
  886 = 'dry'
  198 = 'Dry'
  258 = 'DryRun'
  654 = 'Error'
  70 = 'In'
  143 = 'LED'
  956 = 'Lin21'
  298 = 'Line1'
  372 = 'Line2'
  137 = 'Line2Dismantling'
  471 = 'Line3'
  302 = 'Line3Dismantling'
  837 = 'Line3Load'
  75 = 'LineAxis'
  817 = 'MachineType:%s'
  850 = 'None'
  492 = 'Operator'
  924 = 'RH200'
  133 = 'Service'
  213 = 'Station'
  58 = 'UnloadElevator'
  405 = 'UnloadElevatorne2'
  418 = 'UnloadUc'
  575 = '空跑'
  943 = '线体2拆解站'
END_TEXTLIST

// ---- VISUs/Ctrl/CtrlLine.TcVIS
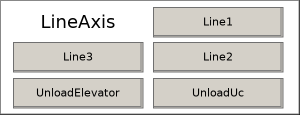
VISUALIZATION CtrlLine  // 300x115
    RoundedRectangle (0,0 300x115)
    Button (153,7 130x30), "Line1"
        OnMouseDown: execute { GVL.arrFbLine[E_Line.Line1].M_Jog(1); }
        OnMouseUp: execute { GVL.arrFbLine[E_Line.Line1].M_Jog(0); }
    Button (153,42 130x30), "Line2"
        OnMouseDown: execute { GVL.arrFbLine[E_Line.Line2].M_Jog(1); }
        OnMouseUp: execute { GVL.arrFbLine[E_Line.Line2].M_Jog(0); }
    Button (13,42 130x30), "Line3"
        OnMouseDown: execute { GVL.arrFbLine[E_Line.Line3].M_Jog(1); }
        OnMouseUp: execute { GVL.arrFbLine[E_Line.Line3].M_Jog(0); }
    Button (153,78 130x30), "UnloadUc"
        OnMouseDown: execute { GVL.arrFbLine[E_Line.UnloadUC].M_Jog(1); }
        OnMouseUp: execute { GVL.arrFbLine[E_Line.UnloadUC].M_Jog(0); }
    Button (13,78 130x30), "UnloadElevator"
        OnMouseDown: execute { GVL.arrFbLine[E_Line.UnloadElevator].M_Jog(1); }
        OnMouseUp: execute { GVL.arrFbLine[E_Line.UnloadElevator].M_Jog(0); }
    Label (13,7 130x30), "LineAxis"
END_VISUALIZATION

// ---- VISUs/Ctrl/CtrlOther.TcVIS
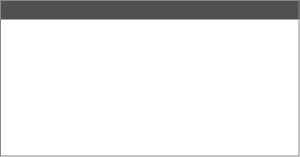
VISUALIZATION CtrlOther  // 300x157
    Rectangle (0,0 300x157)
    Rectangle (0,0 300x19)
END_VISUALIZATION

// ---- VISUs/Ctrl/CtrlOutput.TcVIS
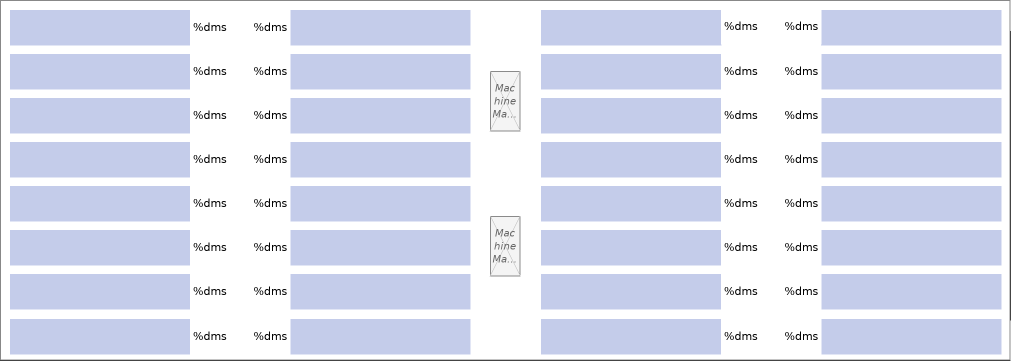
VISUALIZATION CtrlOutput  // 1011x361
VAR_INPUT
	In:						POINTER TO BOOL;
	SizeIn:					DINT;
	Enable:					BOOL;// 是否启用强制功能
	Ton:					POINTER TO UINT;// 延迟区域
	In_S:					POINTER TO BOOL;
END_VAR
VAR
	_pageCount:				INT;
	_index:					INT;
END_VAR
    RoundedRectangle (0,0 1010x115)
    RoundedRectangle (0,246 1010x115)
    Rectangle (0,52 1010x268)
    Line (1010,31) (1010,320)
    Line (0,33) (0,332)
    Image (490,71 30x60), image: MachineManage.ImagePool.prev
        OnMouseDown: execute {
            IF _index-32>=0 THEN
            	_index:=_index-32;
            END_IF
        }
    Image (490,216 30x60), image: MachineManage.ImagePool.next
        OnMouseClick: execute {
            IF SizeIn>_index+32 THEN
            	_index:=_index+32;
            END_IF
        }
    RoundedRectangle (10,10 180x35), colour toggle: In[_index], invisible if: SizeIn<=_index, input disabled if: In_S[_index], text list: 'OutputText', text index: _index
        OnMouseClick: execute {
            IF Enable AND SizeIn>_index THEN
            	In[_index]:=NOT In[_index];
            END_IF;
        }
    RoundedRectangle (10,54 180x35), colour toggle: In[1+_index], invisible if: SizeIn<= 1+_index, input disabled if: In_S[1+_index], text list: 'OutputText', text index: 1+_index
        OnMouseClick: execute {
            IF Enable AND SizeIn>_index+1 THEN
            	In[_index+1]:=NOT In[_index+1];
            END_IF;
        }
    RoundedRectangle (10,98 180x35), colour toggle: In[2+_index], invisible if: SizeIn<= 2+_index, input disabled if: In_S[2+_index], text list: 'OutputText', text index: 2+_index
        OnMouseClick: execute {
            IF Enable AND SizeIn>_index+2 THEN
            	In[_index+2]:=NOT In[_index+2];
            END_IF;
        }
    RoundedRectangle (10,142 180x35), colour toggle: In[3+_index], invisible if: SizeIn<=3+_index, input disabled if: In_S[3+_index], text list: 'OutputText', text index: 3+_index
        OnMouseClick: execute {
            IF Enable AND SizeIn>_index+3 THEN
            	In[_index+3]:=NOT In[_index+3];
            END_IF;
        }
    RoundedRectangle (10,186 180x35), colour toggle: In[_index+4], invisible if: SizeIn<=_index+4, input disabled if: In_S[_index+4], text list: 'OutputText', text index: _index+4
        OnMouseClick: execute {
            IF Enable AND SizeIn>_index+4 THEN
            	In[_index+4]:=NOT In[_index+4];
            END_IF;
        }
    RoundedRectangle (10,230 180x35), colour toggle: In[_index+5], invisible if: SizeIn<=_index+5, input disabled if: In_S[_index+5], text list: 'OutputText', text index: _index+5
        OnMouseClick: execute {
            IF Enable AND SizeIn>_index+5 THEN
            	In[_index+5]:=NOT In[_index+5];
            END_IF;
        }
    RoundedRectangle (10,274 180x35), colour toggle: In[_index+6], invisible if: SizeIn<=_index+6, input disabled if: In_S[_index+6], text list: 'OutputText', text index: _index+6
        OnMouseClick: execute {
            IF Enable AND SizeIn>_index+6 THEN
            	In[_index+6]:=NOT In[_index+6];
            END_IF;
        }
    RoundedRectangle (10,319 180x35), colour toggle: In[_index+7], invisible if: SizeIn<=_index+7, input disabled if: In_S[_index+7], text list: 'OutputText', text index: _index+7
        OnMouseClick: execute {
            IF Enable AND SizeIn>_index+7 THEN
            	In[_index+7]:=NOT In[_index+7];
            END_IF;
        }
    RoundedRectangle (290,10 180x35), colour toggle: In[_index+8], invisible if: SizeIn<=_index+8, input disabled if: In_S[_index+8], text list: 'OutputText', text index: _index+8
        OnMouseClick: execute {
            IF Enable AND SizeIn>_index+8 THEN
            	In[_index+8]:=NOT In[_index+8];
            END_IF;
        }
    RoundedRectangle (290,54 180x35), colour toggle: In[_index+9], invisible if: SizeIn<=_index+9, input disabled if: In_S[_index+9], text list: 'OutputText', text index: _index+9
        OnMouseClick: execute {
            IF Enable AND SizeIn>_index+9 THEN
            	In[_index+9]:=NOT In[_index+9];
            END_IF;
        }
    RoundedRectangle (290,98 180x35), colour toggle: In[_index+10], invisible if: SizeIn<=_index+10, input disabled if: In_S[_index+10], text list: 'OutputText', text index: _index+10
        OnMouseClick: execute {
            IF Enable AND SizeIn>_index+10 THEN
            	In[_index+10]:=NOT In[_index+10];
            END_IF;
        }
    RoundedRectangle (290,142 180x35), colour toggle: In[_index+11], invisible if: SizeIn<=_index+11, input disabled if: In_S[_index+11], text list: 'OutputText', text index: _index+11
        OnMouseClick: execute {
            IF Enable AND SizeIn>_index+11 THEN
            	In[_index+11]:=NOT In[_index+11];
            END_IF;
        }
    RoundedRectangle (290,186 180x35), colour toggle: In[_index+12], invisible if: SizeIn<=_index+12, input disabled if: In_S[_index+12], text list: 'OutputText', text index: _index+12
        OnMouseClick: execute {
            IF Enable AND SizeIn>_index+12 THEN
            	In[_index+12]:=NOT In[_index+12];
            END_IF;
        }
    RoundedRectangle (290,230 180x35), colour toggle: In[_index+13], invisible if: SizeIn<=_index+13, input disabled if: In_S[_index+13], text list: 'OutputText', text index: _index+13
        OnMouseClick: execute {
            IF Enable AND SizeIn>_index+13 THEN
            	In[_index+13]:=NOT In[_index+13];
            END_IF;
        }
    RoundedRectangle (290,274 180x35), colour toggle: In[_index+14], invisible if: SizeIn<=_index+14, input disabled if: In_S[_index+14], text list: 'OutputText', text index: _index+14
        OnMouseClick: execute {
            IF Enable AND SizeIn>_index+14 THEN
            	In[_index+14]:=NOT In[_index+14];
            END_IF;
        }
    RoundedRectangle (290,319 180x35), colour toggle: In[_index+15], invisible if: SizeIn<=_index+15, input disabled if: In_S[_index+15], text list: 'OutputText', text index: _index+15
        OnMouseClick: execute {
            IF Enable AND SizeIn>_index+15 THEN
            	In[_index+15]:=NOT In[_index+15];
            END_IF;
        }
    RoundedRectangle (541,10 180x35), colour toggle: In[_index+16], invisible if: SizeIn<=_index+16, input disabled if: In_S[_index+16], text list: 'OutputText', text index: _index+16
        OnMouseClick: execute {
            IF Enable AND SizeIn>_index+16 THEN
            	In[_index+16]:=NOT In[_index+16];
            END_IF;
        }
    RoundedRectangle (541,54 180x35), colour toggle: In[_index+17], invisible if: SizeIn<=_index+17, input disabled if: In_S[_index+17], text list: 'OutputText', text index: _index+17
        OnMouseClick: execute {
            IF Enable AND SizeIn>_index+17 THEN
            	In[_index+17]:=NOT In[_index+17];
            END_IF;
        }
    RoundedRectangle (541,98 180x35), colour toggle: In[_index+18], invisible if: SizeIn<=_index+18, input disabled if: In_S[_index+18], text list: 'OutputText', text index: _index+18
        OnMouseClick: execute {
            IF Enable AND SizeIn>_index+18 THEN
            	In[_index+18]:=NOT In[_index+18];
            END_IF;
        }
    RoundedRectangle (541,142 180x35), colour toggle: In[_index+19], invisible if: SizeIn<=_index+19, input disabled if: In_S[_index+19], text list: 'OutputText', text index: _index+19
        OnMouseClick: execute {
            IF Enable AND SizeIn>_index+19 THEN
            	In[_index+19]:=NOT In[_index+19];
            END_IF;
        }
    RoundedRectangle (541,186 180x35), colour toggle: In[_index+20], invisible if: SizeIn<=_index+20, input disabled if: In_S[_index+20], text list: 'OutputText', text index: _index+20
        OnMouseClick: execute {
            IF Enable AND SizeIn>_index+20 THEN
            	In[_index+20]:=NOT In[_index+20];
            END_IF;
        }
    RoundedRectangle (541,230 180x35), colour toggle: In[_index+21], invisible if: SizeIn<=_index+21, input disabled if: In_S[_index+21], text list: 'OutputText', text index: _index+21
        OnMouseClick: execute {
            IF Enable AND SizeIn>_index+21 THEN
            	In[_index+21]:=NOT In[_index+21];
            END_IF;
        }
    RoundedRectangle (541,274 180x35), colour toggle: In[_index+22], invisible if: SizeIn<=_index+22, input disabled if: In_S[_index+22], text list: 'OutputText', text index: _index+22
        OnMouseClick: execute {
            IF Enable AND SizeIn>_index+22 THEN
            	In[_index+22]:=NOT In[_index+22];
            END_IF;
        }
    RoundedRectangle (541,319 180x35), colour toggle: In[_index+23], invisible if: SizeIn<=_index+23, input disabled if: In_S[_index+23], text list: 'OutputText', text index: _index+23
        OnMouseClick: execute {
            IF Enable AND SizeIn>_index+23 THEN
            	In[_index+23]:=NOT In[_index+23];
            END_IF;
        }
    RoundedRectangle (821,10 180x35), colour toggle: In[_index+24], invisible if: SizeIn<=_index+24, input disabled if: In_S[_index+24], text list: 'OutputText', text index: _index+24
        OnMouseClick: execute {
            IF Enable AND SizeIn>_index+24 THEN
            	In[_index+24]:=NOT In[_index+24];
            END_IF;
        }
    RoundedRectangle (821,54 180x35), colour toggle: In[_index+25], invisible if: SizeIn<=_index+25, input disabled if: In_S[_index+25], text list: 'OutputText', text index: _index+25
        OnMouseClick: execute {
            IF Enable AND SizeIn>_index+25 THEN
            	In[_index+25]:=NOT In[_index+25];
            END_IF;
        }
    RoundedRectangle (821,98 180x35), colour toggle: In[_index+26], invisible if: SizeIn<=_index+26, input disabled if: In_S[_index+26], text list: 'OutputText', text index: _index+26
        OnMouseClick: execute {
            IF Enable AND SizeIn>_index+26 THEN
            	In[_index+26]:=NOT In[_index+26];
            END_IF;
        }
    RoundedRectangle (821,142 180x35), colour toggle: In[_index+27], invisible if: SizeIn<=_index+27, input disabled if: In_S[_index+27], text list: 'OutputText', text index: _index+27
        OnMouseClick: execute {
            IF Enable AND SizeIn>_index+27 THEN
            	In[_index+27]:=NOT In[_index+27];
            END_IF;
        }
    RoundedRectangle (821,186 180x35), colour toggle: In[_index+28], invisible if: SizeIn<=_index+28, input disabled if: In_S[_index+28], text list: 'OutputText', text index: _index+28
        OnMouseClick: execute {
            IF Enable AND SizeIn>_index+28 THEN
            	In[_index+28]:=NOT In[_index+28];
            END_IF;
        }
    RoundedRectangle (821,230 180x35), colour toggle: In[_index+29], invisible if: SizeIn<=_index+29, input disabled if: In_S[_index+29], text list: 'OutputText', text index: _index+29
        OnMouseClick: execute {
            IF Enable AND SizeIn>_index+29 THEN
            	In[_index+29]:=NOT In[_index+29];
            END_IF;
        }
    RoundedRectangle (821,274 180x35), colour toggle: In[_index+30], invisible if: SizeIn<=_index+30, input disabled if: In_S[_index+30], text list: 'OutputText', text index: _index+30
        OnMouseClick: execute {
            IF Enable AND SizeIn>_index+30 THEN
            	In[_index+30]:=NOT In[_index+30];
            END_IF;
        }
    RoundedRectangle (821,319 180x35), colour toggle: In[_index+31], invisible if: SizeIn<=_index+31, input disabled if: In_S[_index+31], text list: 'OutputText', text index: _index+31
        OnMouseClick: execute {
            IF Enable AND SizeIn>_index+31 THEN
            	In[_index+31]:=NOT In[_index+31];
            END_IF;
        }
    Rectangle (190,10 50x35), "%dms", text variable: Ton[_index], invisible if: SizeIn<=_index
        OnMouseClick: write the text variable via Default, min 0
    Rectangle (240,10 50x35), "%dms", text variable: Ton[_index+8], invisible if: SizeIn<=_index+8
        OnMouseClick: write the text variable via Default, min 0
    Rectangle (190,54 50x35), "%dms", text variable: Ton[_index+1], invisible if: SizeIn<=_index+1
        OnMouseClick: write the text variable via Default, min 0
    Rectangle (240,54 50x35), "%dms", text variable: Ton[_index+9], invisible if: SizeIn<=_index+9
        OnMouseClick: write the text variable via Default, min 0
    Rectangle (190,98 50x35), "%dms", text variable: Ton[_index+2], invisible if: SizeIn<=_index+2
        OnMouseClick: write the text variable via Default, min 0
    Rectangle (240,98 50x35), "%dms", text variable: Ton[_index+10], invisible if: SizeIn<=_index+10
        OnMouseClick: write the text variable via Default, min 0
    Rectangle (190,142 50x35), "%dms", text variable: Ton[_index+3], invisible if: SizeIn<=_index+3
        OnMouseClick: write the text variable via Default, min 0
    Rectangle (240,142 50x35), "%dms", text variable: Ton[_index+11], invisible if: SizeIn<=_index+11
        OnMouseClick: write the text variable via Default, min 0
    Rectangle (190,186 50x35), "%dms", text variable: Ton[_index+4], invisible if: SizeIn<=_index+4
        OnMouseClick: write the text variable via Default, min 0
    Rectangle (240,186 50x35), "%dms", text variable: Ton[_index+12], invisible if: SizeIn<=_index+12
        OnMouseClick: write the text variable via Default, min 0
    Rectangle (190,230 50x35), "%dms", text variable: Ton[_index+5], invisible if: SizeIn<=_index+5
        OnMouseClick: write the text variable via Default, min 0
    Rectangle (240,230 50x35), "%dms", text variable: Ton[_index+13], invisible if: SizeIn<=_index+13
        OnMouseClick: write the text variable via Default, min 0
    Rectangle (190,274 50x35), "%dms", text variable: Ton[_index+6], invisible if: SizeIn<=_index+6
        OnMouseClick: write the text variable via Default, min 0
    Rectangle (240,274 50x35), "%dms", text variable: Ton[_index+14], invisible if: SizeIn<=_index+14
        OnMouseClick: write the text variable via Default, min 0
    Rectangle (190,319 50x35), "%dms", text variable: Ton[_index+7], invisible if: SizeIn<=_index+7
        OnMouseClick: write the text variable via Default, min 0
    Rectangle (240,319 50x35), "%dms", text variable: Ton[_index+15], invisible if: SizeIn<=_index+15
        OnMouseClick: write the text variable via Default, min 0
    Rectangle (721,9 50x35), "%dms", text variable: Ton[_index+16], invisible if: SizeIn<=_index+16
        OnMouseClick: write the text variable via Default, min 0
    Rectangle (771,9 50x35), "%dms", text variable: Ton[_index+24], invisible if: SizeIn<=_index+24
        OnMouseClick: write the text variable via Default, min 0
    Rectangle (721,54 50x35), "%dms", text variable: Ton[_index+17], invisible if: SizeIn<=_index+17
        OnMouseClick: write the text variable via Default, min 0
    Rectangle (771,54 50x35), "%dms", text variable: Ton[_index+25], invisible if: SizeIn<=_index+25
        OnMouseClick: write the text variable via Default, min 0
    Rectangle (721,98 50x35), "%dms", text variable: Ton[_index+18], invisible if: SizeIn<=_index+18
        OnMouseClick: write the text variable via Default, min 0
    Rectangle (771,98 50x35), "%dms", text variable: Ton[_index+26], invisible if: SizeIn<=_index+26
        OnMouseClick: write the text variable via Default, min 0
    Rectangle (721,142 50x35), "%dms", text variable: Ton[_index+19], invisible if: SizeIn<=_index+19
        OnMouseClick: write the text variable via Default, min 0
    Rectangle (771,142 50x35), "%dms", text variable: Ton[_index+27], invisible if: SizeIn<=_index+27
        OnMouseClick: write the text variable via Default, min 0
    Rectangle (721,186 50x35), "%dms", text variable: Ton[_index+20], invisible if: SizeIn<=_index+20
        OnMouseClick: write the text variable via Default, min 0
    Rectangle (771,186 50x35), "%dms", text variable: Ton[_index+28], invisible if: SizeIn<=_index+28
        OnMouseClick: write the text variable via Default, min 0
    Rectangle (721,230 50x35), "%dms", text variable: Ton[_index+21], invisible if: SizeIn<=_index+21
        OnMouseClick: write the text variable via Default, min 0
    Rectangle (771,230 50x35), "%dms", text variable: Ton[_index+29], invisible if: SizeIn<=_index+29
        OnMouseClick: write the text variable via Default, min 0
    Rectangle (721,274 50x35), "%dms", text variable: Ton[_index+22], invisible if: SizeIn<=_index+22
        OnMouseClick: write the text variable via Default, min 0
    Rectangle (771,274 50x35), "%dms", text variable: Ton[_index+30], invisible if: SizeIn<=_index+30
        OnMouseClick: write the text variable via Default, min 0
    Rectangle (721,319 50x35), "%dms", text variable: Ton[_index+23], invisible if: SizeIn<=_index+23
        OnMouseClick: write the text variable via Default, min 0
    Rectangle (771,319 50x35), "%dms", text variable: Ton[_index+31], invisible if: SizeIn<=_index+31
        OnMouseClick: write the text variable via Default, min 0
END_VISUALIZATION

// ---- VISUs/Ctrl/CtrlInput.TcVIS
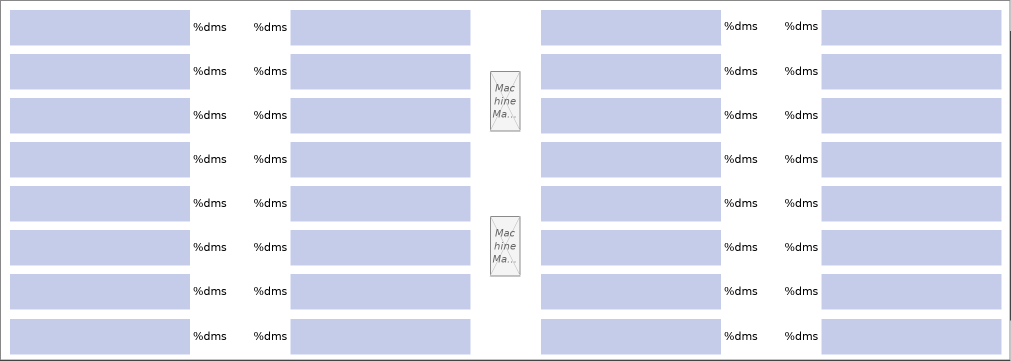
VISUALIZATION CtrlInput  // 1011x361
VAR_INPUT
	In:						POINTER TO BOOL;
	SizeIn:					DINT;
	Enable:					BOOL;// 是否启用强制功能
	Ton:					POINTER TO UINT;// 延迟区域
	In_S:					POINTER TO BOOL;
END_VAR
VAR
	_pageCount:				INT;
	_index:					INT;
END_VAR
    RoundedRectangle (0,0 1010x115)
    RoundedRectangle (0,246 1010x115)
    Rectangle (0,52 1010x268)
    Line (1010,31) (1010,320)
    Line (0,33) (0,332)
    Image (490,71 30x60), image: MachineManage.ImagePool.prev
        OnMouseDown: execute {
            IF _index-32>=0 THEN
            	_index:=_index-32;
            END_IF
        }
    Image (490,216 30x60), image: MachineManage.ImagePool.next
        OnMouseClick: execute {
            IF SizeIn>_index+32 THEN
            	_index:=_index+32;
            END_IF
        }
    RoundedRectangle (10,10 180x35), colour toggle: In[_index], invisible if: SizeIn<=_index, input disabled if: In_S[_index], text list: 'InputText', text index: _index
        OnMouseClick: execute {
            IF Enable AND SizeIn>_index THEN
            	In[_index]:=NOT In[_index];
            END_IF;
        }
    RoundedRectangle (10,54 180x35), colour toggle: In[1+_index], invisible if: SizeIn<= 1+_index, input disabled if: In_S[1+_index], text list: 'InputText', text index: 1+_index
        OnMouseClick: execute {
            IF Enable AND SizeIn>_index+1 THEN
            	In[_index+1]:=NOT In[_index+1];
            END_IF;
        }
    RoundedRectangle (10,98 180x35), colour toggle: In[2+_index], invisible if: SizeIn<= 2+_index, input disabled if: In_S[2+_index], text list: 'InputText', text index: 2+_index
        OnMouseClick: execute {
            IF Enable AND SizeIn>_index+2 THEN
            	In[_index+2]:=NOT In[_index+2];
            END_IF;
        }
    RoundedRectangle (10,142 180x35), colour toggle: In[3+_index], invisible if: SizeIn<=3+_index, input disabled if: In_S[3+_index], text list: 'InputText', text index: 3+_index
        OnMouseClick: execute {
            IF Enable AND SizeIn>_index+3 THEN
            	In[_index+3]:=NOT In[_index+3];
            END_IF;
        }
    RoundedRectangle (10,186 180x35), colour toggle: In[_index+4], invisible if: SizeIn<=_index+4, input disabled if: In_S[_index+4], text list: 'InputText', text index: _index+4
        OnMouseClick: execute {
            IF Enable AND SizeIn>_index+4 THEN
            	In[_index+4]:=NOT In[_index+4];
            END_IF;
        }
    RoundedRectangle (10,230 180x35), colour toggle: In[_index+5], invisible if: SizeIn<=_index+5, input disabled if: In_S[_index+5], text list: 'InputText', text index: _index+5
        OnMouseClick: execute {
            IF Enable AND SizeIn>_index+5 THEN
            	In[_index+5]:=NOT In[_index+5];
            END_IF;
        }
    RoundedRectangle (10,274 180x35), colour toggle: In[_index+6], invisible if: SizeIn<=_index+6, input disabled if: In_S[_index+6], text list: 'InputText', text index: _index+6
        OnMouseClick: execute {
            IF Enable AND SizeIn>_index+6 THEN
            	In[_index+6]:=NOT In[_index+6];
            END_IF;
        }
    RoundedRectangle (10,319 180x35), colour toggle: In[_index+7], invisible if: SizeIn<=_index+7, input disabled if: In_S[_index+7], text list: 'InputText', text index: _index+7
        OnMouseClick: execute {
            IF Enable AND SizeIn>_index+7 THEN
            	In[_index+7]:=NOT In[_index+7];
            END_IF;
        }
    RoundedRectangle (290,10 180x35), colour toggle: In[_index+8], invisible if: SizeIn<=_index+8, input disabled if: In_S[_index+8], text list: 'InputText', text index: _index+8
        OnMouseClick: execute {
            IF Enable AND SizeIn>_index+8 THEN
            	In[_index+8]:=NOT In[_index+8];
            END_IF;
        }
    RoundedRectangle (290,54 180x35), colour toggle: In[_index+9], invisible if: SizeIn<=_index+9, input disabled if: In_S[_index+9], text list: 'InputText', text index: _index+9
        OnMouseClick: execute {
            IF Enable AND SizeIn>_index+9 THEN
            	In[_index+9]:=NOT In[_index+9];
            END_IF;
        }
    RoundedRectangle (290,98 180x35), colour toggle: In[_index+10], invisible if: SizeIn<=_index+10, input disabled if: In_S[_index+10], text list: 'InputText', text index: _index+10
        OnMouseClick: execute {
            IF Enable AND SizeIn>_index+10 THEN
            	In[_index+10]:=NOT In[_index+10];
            END_IF;
        }
    RoundedRectangle (290,142 180x35), colour toggle: In[_index+11], invisible if: SizeIn<=_index+11, input disabled if: In_S[_index+11], text list: 'InputText', text index: _index+11
        OnMouseClick: execute {
            IF Enable AND SizeIn>_index+11 THEN
            	In[_index+11]:=NOT In[_index+11];
            END_IF;
        }
    RoundedRectangle (290,186 180x35), colour toggle: In[_index+12], invisible if: SizeIn<=_index+12, input disabled if: In_S[_index+12], text list: 'InputText', text index: _index+12
        OnMouseClick: execute {
            IF Enable AND SizeIn>_index+12 THEN
            	In[_index+12]:=NOT In[_index+12];
            END_IF;
        }
    RoundedRectangle (290,230 180x35), colour toggle: In[_index+13], invisible if: SizeIn<=_index+13, input disabled if: In_S[_index+13], text list: 'InputText', text index: _index+13
        OnMouseClick: execute {
            IF Enable AND SizeIn>_index+13 THEN
            	In[_index+13]:=NOT In[_index+13];
            END_IF;
        }
    RoundedRectangle (290,274 180x35), colour toggle: In[_index+14], invisible if: SizeIn<=_index+14, input disabled if: In_S[_index+14], text list: 'InputText', text index: _index+14
        OnMouseClick: execute {
            IF Enable AND SizeIn>_index+14 THEN
            	In[_index+14]:=NOT In[_index+14];
            END_IF;
        }
    RoundedRectangle (290,319 180x35), colour toggle: In[_index+15], invisible if: SizeIn<=_index+15, input disabled if: In_S[_index+15], text list: 'InputText', text index: _index+15
        OnMouseClick: execute {
            IF Enable AND SizeIn>_index+15 THEN
            	In[_index+15]:=NOT In[_index+15];
            END_IF;
        }
    RoundedRectangle (541,10 180x35), colour toggle: In[_index+16], invisible if: SizeIn<=_index+16, input disabled if: In_S[_index+16], text list: 'InputText', text index: _index+16
        OnMouseClick: execute {
            IF Enable AND SizeIn>_index+16 THEN
            	In[_index+16]:=NOT In[_index+16];
            END_IF;
        }
    RoundedRectangle (541,54 180x35), colour toggle: In[_index+17], invisible if: SizeIn<=_index+17, input disabled if: In_S[_index+17], text list: 'InputText', text index: _index+17
        OnMouseClick: execute {
            IF Enable AND SizeIn>_index+17 THEN
            	In[_index+17]:=NOT In[_index+17];
            END_IF;
        }
    RoundedRectangle (541,98 180x35), colour toggle: In[_index+18], invisible if: SizeIn<=_index+18, input disabled if: In_S[_index+18], text list: 'InputText', text index: _index+18
        OnMouseClick: execute {
            IF Enable AND SizeIn>_index+18 THEN
            	In[_index+18]:=NOT In[_index+18];
            END_IF;
        }
    RoundedRectangle (541,142 180x35), colour toggle: In[_index+19], invisible if: SizeIn<=_index+19, input disabled if: In_S[_index+19], text list: 'InputText', text index: _index+19
        OnMouseClick: execute {
            IF Enable AND SizeIn>_index+19 THEN
            	In[_index+19]:=NOT In[_index+19];
            END_IF;
        }
    RoundedRectangle (541,186 180x35), colour toggle: In[_index+20], invisible if: SizeIn<=_index+20, input disabled if: In_S[_index+20], text list: 'InputText', text index: _index+20
        OnMouseClick: execute {
            IF Enable AND SizeIn>_index+20 THEN
            	In[_index+20]:=NOT In[_index+20];
            END_IF;
        }
    RoundedRectangle (541,230 180x35), colour toggle: In[_index+21], invisible if: SizeIn<=_index+21, input disabled if: In_S[_index+21], text list: 'InputText', text index: _index+21
        OnMouseClick: execute {
            IF Enable AND SizeIn>_index+21 THEN
            	In[_index+21]:=NOT In[_index+21];
            END_IF;
        }
    RoundedRectangle (541,274 180x35), colour toggle: In[_index+22], invisible if: SizeIn<=_index+22, input disabled if: In_S[_index+22], text list: 'InputText', text index: _index+22
        OnMouseClick: execute {
            IF Enable AND SizeIn>_index+22 THEN
            	In[_index+22]:=NOT In[_index+22];
            END_IF;
        }
    RoundedRectangle (541,319 180x35), colour toggle: In[_index+23], invisible if: SizeIn<=_index+23, input disabled if: In_S[_index+23], text list: 'InputText', text index: _index+23
        OnMouseClick: execute {
            IF Enable AND SizeIn>_index+23 THEN
            	In[_index+23]:=NOT In[_index+23];
            END_IF;
        }
    RoundedRectangle (821,10 180x35), colour toggle: In[_index+24], invisible if: SizeIn<=_index+24, input disabled if: In_S[_index+24], text list: 'InputText', text index: _index+24
        OnMouseClick: execute {
            IF Enable AND SizeIn>_index+24 THEN
            	In[_index+24]:=NOT In[_index+24];
            END_IF;
        }
    RoundedRectangle (821,54 180x35), colour toggle: In[_index+25], invisible if: SizeIn<=_index+25, input disabled if: In_S[_index+25], text list: 'InputText', text index: _index+25
        OnMouseClick: execute {
            IF Enable AND SizeIn>_index+25 THEN
            	In[_index+25]:=NOT In[_index+25];
            END_IF;
        }
    RoundedRectangle (821,98 180x35), colour toggle: In[_index+26], invisible if: SizeIn<=_index+26, input disabled if: In_S[_index+26], text list: 'InputText', text index: _index+26
        OnMouseClick: execute {
            IF Enable AND SizeIn>_index+26 THEN
            	In[_index+26]:=NOT In[_index+26];
            END_IF;
        }
    RoundedRectangle (821,142 180x35), colour toggle: In[_index+27], invisible if: SizeIn<=_index+27, input disabled if: In_S[_index+27], text list: 'InputText', text index: _index+27
        OnMouseClick: execute {
            IF Enable AND SizeIn>_index+27 THEN
            	In[_index+27]:=NOT In[_index+27];
            END_IF;
        }
    RoundedRectangle (821,186 180x35), colour toggle: In[_index+28], invisible if: SizeIn<=_index+28, input disabled if: In_S[_index+28], text list: 'InputText', text index: _index+28
        OnMouseClick: execute {
            IF Enable AND SizeIn>_index+28 THEN
            	In[_index+28]:=NOT In[_index+28];
            END_IF;
        }
    RoundedRectangle (821,230 180x35), colour toggle: In[_index+29], invisible if: SizeIn<=_index+29, input disabled if: In_S[_index+29], text list: 'InputText', text index: _index+29
        OnMouseClick: execute {
            IF Enable AND SizeIn>_index+29 THEN
            	In[_index+29]:=NOT In[_index+29];
            END_IF;
        }
    RoundedRectangle (821,274 180x35), colour toggle: In[_index+30], invisible if: SizeIn<=_index+30, input disabled if: In_S[_index+30], text list: 'InputText', text index: _index+30
        OnMouseClick: execute {
            IF Enable AND SizeIn>_index+30 THEN
            	In[_index+30]:=NOT In[_index+30];
            END_IF;
        }
    RoundedRectangle (821,319 180x35), colour toggle: In[_index+31], invisible if: SizeIn<=_index+31, input disabled if: In_S[_index+31], text list: 'InputText', text index: _index+31
        OnMouseClick: execute {
            IF Enable AND SizeIn>_index+31 THEN
            	In[_index+31]:=NOT In[_index+31];
            END_IF;
        }
    Rectangle (190,10 50x35), "%dms", text variable: Ton[_index], invisible if: SizeIn<=_index
        OnMouseClick: write the text variable via Default, min 0
    Rectangle (240,10 50x35), "%dms", text variable: Ton[_index+8], invisible if: SizeIn<=_index+8
        OnMouseClick: write the text variable via Default, min 0
    Rectangle (190,54 50x35), "%dms", text variable: Ton[_index+1], invisible if: SizeIn<=_index+1
        OnMouseClick: write the text variable via Default, min 0
    Rectangle (240,54 50x35), "%dms", text variable: Ton[_index+9], invisible if: SizeIn<=_index+9
        OnMouseClick: write the text variable via Default, min 0
    Rectangle (190,98 50x35), "%dms", text variable: Ton[_index+2], invisible if: SizeIn<=_index+2
        OnMouseClick: write the text variable via Default, min 0
    Rectangle (240,98 50x35), "%dms", text variable: Ton[_index+10], invisible if: SizeIn<=_index+10
        OnMouseClick: write the text variable via Default, min 0
    Rectangle (190,142 50x35), "%dms", text variable: Ton[_index+3], invisible if: SizeIn<=_index+3
        OnMouseClick: write the text variable via Default, min 0
    Rectangle (240,142 50x35), "%dms", text variable: Ton[_index+11], invisible if: SizeIn<=_index+11
        OnMouseClick: write the text variable via Default, min 0
    Rectangle (190,186 50x35), "%dms", text variable: Ton[_index+4], invisible if: SizeIn<=_index+4
        OnMouseClick: write the text variable via Default, min 0
    Rectangle (240,186 50x35), "%dms", text variable: Ton[_index+12], invisible if: SizeIn<=_index+12
        OnMouseClick: write the text variable via Default, min 0
    Rectangle (190,230 50x35), "%dms", text variable: Ton[_index+5], invisible if: SizeIn<=_index+5
        OnMouseClick: write the text variable via Default, min 0
    Rectangle (240,230 50x35), "%dms", text variable: Ton[_index+13], invisible if: SizeIn<=_index+13
        OnMouseClick: write the text variable via Default, min 0
    Rectangle (190,274 50x35), "%dms", text variable: Ton[_index+6], invisible if: SizeIn<=_index+6
        OnMouseClick: write the text variable via Default, min 0
    Rectangle (240,274 50x35), "%dms", text variable: Ton[_index+14], invisible if: SizeIn<=_index+14
        OnMouseClick: write the text variable via Default, min 0
    Rectangle (190,319 50x35), "%dms", text variable: Ton[_index+7], invisible if: SizeIn<=_index+7
        OnMouseClick: write the text variable via Default, min 0
    Rectangle (240,319 50x35), "%dms", text variable: Ton[_index+15], invisible if: SizeIn<=_index+15
        OnMouseClick: write the text variable via Default, min 0
    Rectangle (721,9 50x35), "%dms", text variable: Ton[_index+16], invisible if: SizeIn<=_index+16
        OnMouseClick: write the text variable via Default, min 0
    Rectangle (771,9 50x35), "%dms", text variable: Ton[_index+24], invisible if: SizeIn<=_index+24
        OnMouseClick: write the text variable via Default, min 0
    Rectangle (721,54 50x35), "%dms", text variable: Ton[_index+17], invisible if: SizeIn<=_index+17
        OnMouseClick: write the text variable via Default, min 0
    Rectangle (771,54 50x35), "%dms", text variable: Ton[_index+25], invisible if: SizeIn<=_index+25
        OnMouseClick: write the text variable via Default, min 0
    Rectangle (721,98 50x35), "%dms", text variable: Ton[_index+18], invisible if: SizeIn<=_index+18
        OnMouseClick: write the text variable via Default, min 0
    Rectangle (771,98 50x35), "%dms", text variable: Ton[_index+26], invisible if: SizeIn<=_index+26
        OnMouseClick: write the text variable via Default, min 0
    Rectangle (721,142 50x35), "%dms", text variable: Ton[_index+19], invisible if: SizeIn<=_index+19
        OnMouseClick: write the text variable via Default, min 0
    Rectangle (771,142 50x35), "%dms", text variable: Ton[_index+27], invisible if: SizeIn<=_index+27
        OnMouseClick: write the text variable via Default, min 0
    Rectangle (721,186 50x35), "%dms", text variable: Ton[_index+20], invisible if: SizeIn<=_index+20
        OnMouseClick: write the text variable via Default, min 0
    Rectangle (771,186 50x35), "%dms", text variable: Ton[_index+28], invisible if: SizeIn<=_index+28
        OnMouseClick: write the text variable via Default, min 0
    Rectangle (721,230 50x35), "%dms", text variable: Ton[_index+21], invisible if: SizeIn<=_index+21
        OnMouseClick: write the text variable via Default, min 0
    Rectangle (771,230 50x35), "%dms", text variable: Ton[_index+29], invisible if: SizeIn<=_index+29
        OnMouseClick: write the text variable via Default, min 0
    Rectangle (721,274 50x35), "%dms", text variable: Ton[_index+22], invisible if: SizeIn<=_index+22
        OnMouseClick: write the text variable via Default, min 0
    Rectangle (771,274 50x35), "%dms", text variable: Ton[_index+30], invisible if: SizeIn<=_index+30
        OnMouseClick: write the text variable via Default, min 0
    Rectangle (721,319 50x35), "%dms", text variable: Ton[_index+23], invisible if: SizeIn<=_index+23
        OnMouseClick: write the text variable via Default, min 0
    Rectangle (771,319 50x35), "%dms", text variable: Ton[_index+31], invisible if: SizeIn<=_index+31
        OnMouseClick: write the text variable via Default, min 0
END_VISUALIZATION

// ---- VISUs/Ctrl/FrameMain.TcVIS
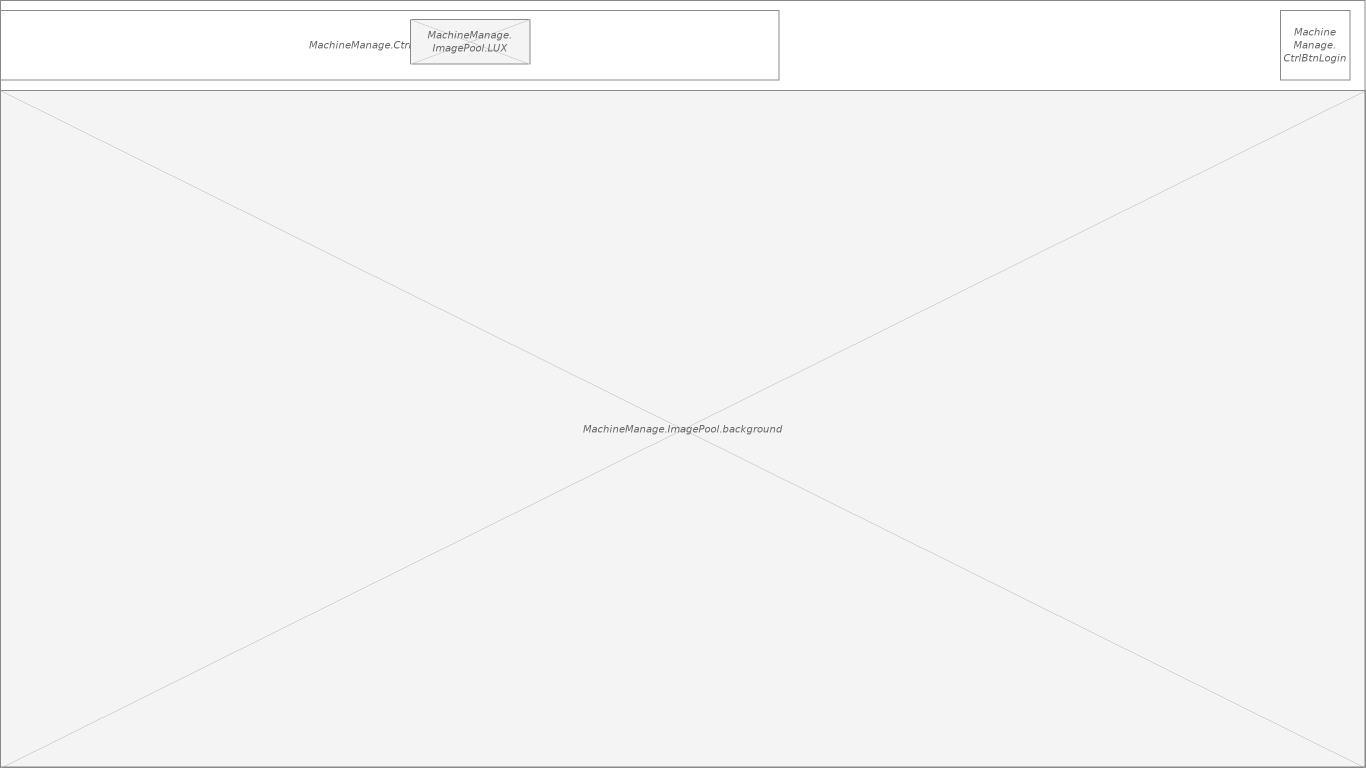
VISUALIZATION FrameMain  // 1366x768
    Frame (0,10 779x70)
        shows MachineManage.CtrlPageSwitch(System := G_stSystem)
    Image (0,90 1366x678), image: MachineManage.ImagePool.background
    Frame (1280,10 70x70)
        shows MachineManage.CtrlBtnLogin()
    Rectangle (422,27 100x30)
    Image (410,19 120x45), image: MachineManage.ImagePool.LUX
END_VISUALIZATION

// ---- VISUs/PageData.TcVIS
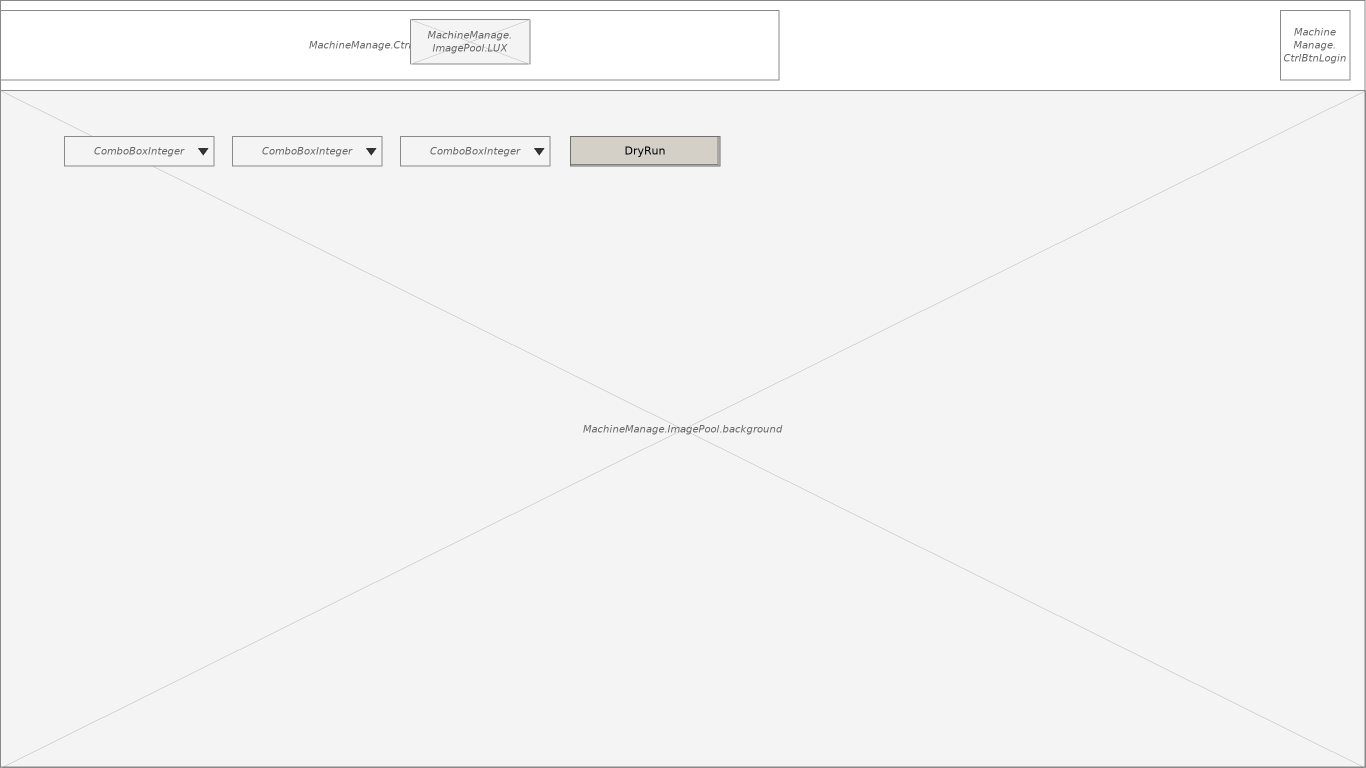
VISUALIZATION PageData  // 1366x768
    Frame (0,0 1366x768)
        shows FrameMain()
    ComboBoxInteger (64,136 150x30), variable: GVL_Data.stRecipe.eLoadClose, text list: 'LineLoadClose'
    ComboBoxInteger (232,136 150x30), variable: GVL_Data.stRecipe.eLineClose, text list: 'LineClose'
    ComboBoxInteger (400,136 150x30), variable: GVL_Data.stRecipe.eLoadPriority, text list: 'LoadPriority'
    Button (570,136 150x30), "DryRun"
        toggle GVL.stSetting.bDryRun
END_VISUALIZATION

// ---- VISUs/PageHome.TcVIS
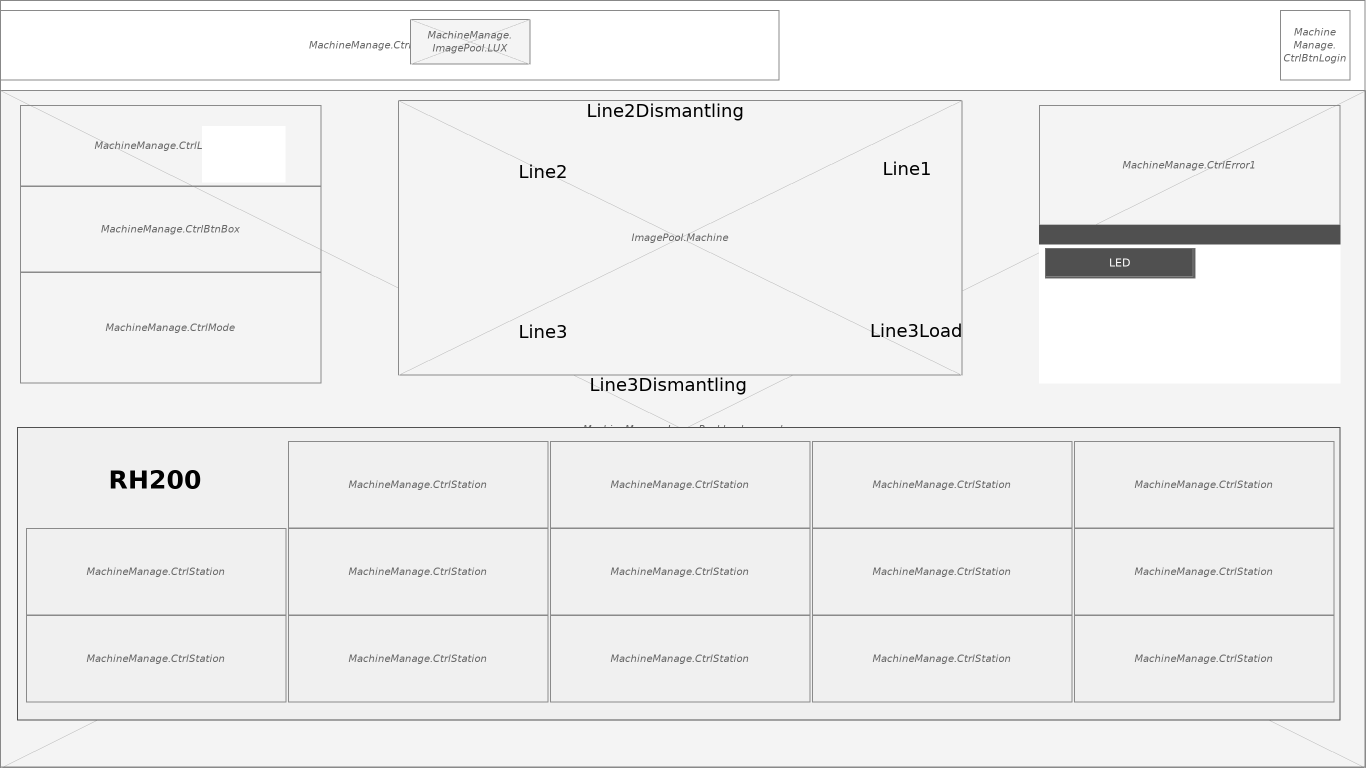
VISUALIZATION PageHome  // 1366x768
    Image (410,98 528x280), image: ImagePool.123
    Frame (0,0 1366x768)
        shows FrameMain()
    Image (398,100 564x275), image: ImagePool.Machine
    Rectangle (17,427 1323x293)
    Frame (20,105 301x81)
        shows MachineManage.CtrlLanguage(System := G_stSystem)
    Frame (20,186 301x86)
        shows MachineManage.CtrlBtnBox(System := G_stSystem)
    Frame (20,272 301x111)
        shows MachineManage.CtrlMode(System := G_stSystem)
    Frame (288,528 260x87)
        shows MachineManage.CtrlStation(System := G_stSystem, Station := G_arrStation[5])
    Frame (550,528 260x87)
        shows MachineManage.CtrlStation(System := G_stSystem, Station := G_arrStation[6])
    Frame (812,528 260x87)
        shows MachineManage.CtrlStation(System := G_stSystem, Station := G_arrStation[7])
    Frame (1074,528 260x87)
        shows MachineManage.CtrlStation(System := G_stSystem, Station := G_arrStation[8])
    Frame (26,615 260x87)
        shows MachineManage.CtrlStation(System := G_stSystem, Station := G_arrStation[9])
    Frame (288,615 260x87)
        shows MachineManage.CtrlStation(System := G_stSystem, Station := G_arrStation[10])
    Frame (550,615 260x87)
        shows MachineManage.CtrlStation(System := G_stSystem, Station := G_arrStation[11])
    Frame (812,615 260x87)
        shows MachineManage.CtrlStation(System := G_stSystem, Station := G_arrStation[12])
    Frame (1074,615 260x87)
        shows MachineManage.CtrlStation(System := G_stSystem, Station := G_arrStation[13])
    Frame (288,441 260x87)
        shows MachineManage.CtrlStation(System := G_stSystem, Station := G_arrStation[0])
    Frame (550,441 260x87)
        shows MachineManage.CtrlStation(System := G_stSystem, Station := G_arrStation[1])
    Frame (812,441 260x87)
        shows MachineManage.CtrlStation(System := G_stSystem, Station := G_arrStation[2])
    Frame (1074,441 260x87)
        shows MachineManage.CtrlStation(System := G_stSystem, Station := G_arrStation[3])
    Frame (26,528 260x87)
        shows MachineManage.CtrlStation(System := G_stSystem, Station := G_arrStation[4])
    Frame (1039,105 301x120)
        shows MachineManage.CtrlError1(System := G_stSystem, Error := G_stError.stNow)
    Frame (1039,225 301x158)
        shows CtrlOther()
    Label (866,154 82x30), "Line1"
    Label (502,157 82x30), "Line2"
    Label (502,317 82x30), "Line3"
    Label (866,316 101x30), "Line3Load"
    Label (583,96 165x30), "Line2Dismantling"
    Label (586,370 165x30), "Line3Dismantling"
    Rectangle (202,126 83x56)
    Rectangle (49,451 212x57), "RH200", text list: 'MachineType', text index: GVL_Data.stRecipe.eMachineType
    Button (1045,248 150x30), "LED"
        toggle GVL.Q.bLED
END_VISUALIZATION

// ---- VISUs/PageMessage.TcVIS
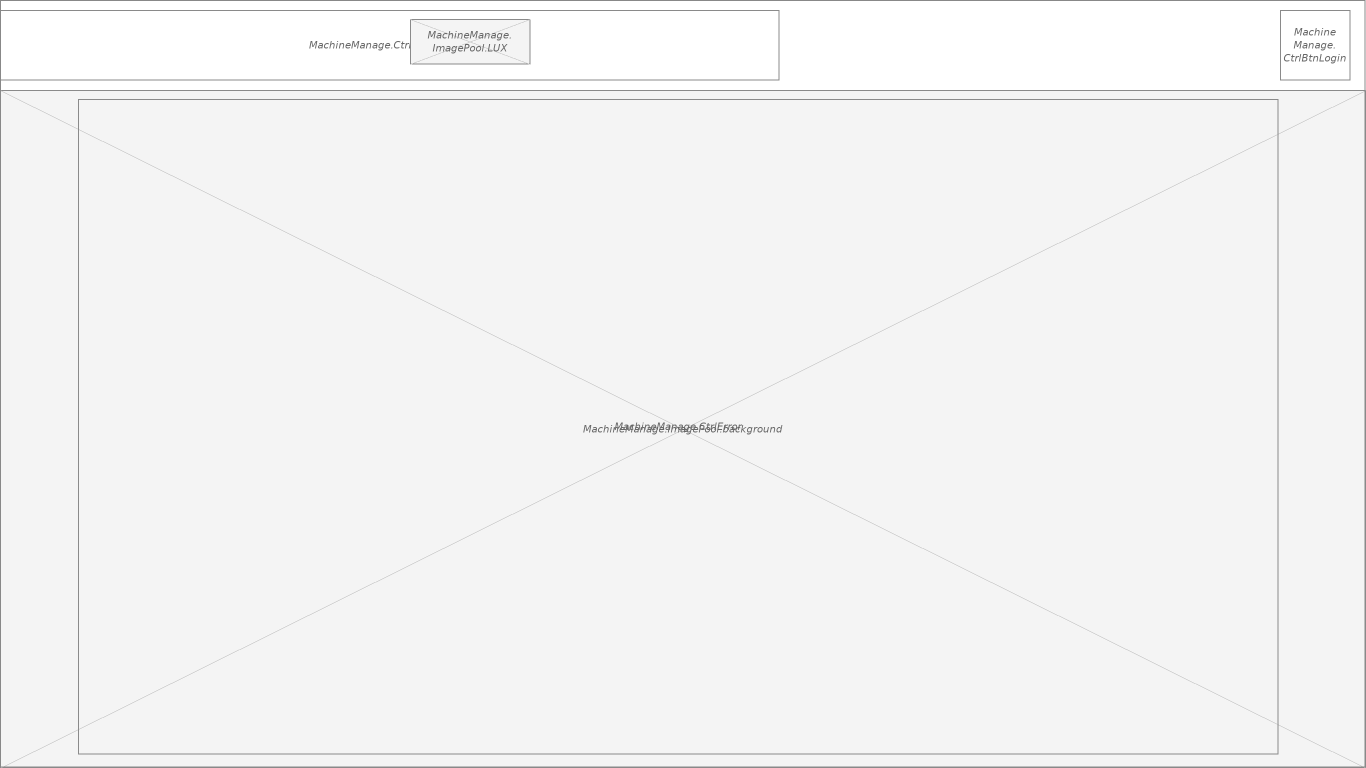
VISUALIZATION PageMessage  // 1366x768
    Frame (0,0 1366x768)
        shows FrameMain()
    Frame (78,99 1200x655)
        shows MachineManage.CtrlError(System := G_stSystem, Error := G_stError)
END_VISUALIZATION

// ---- VISUs/PageMonitor.TcVIS
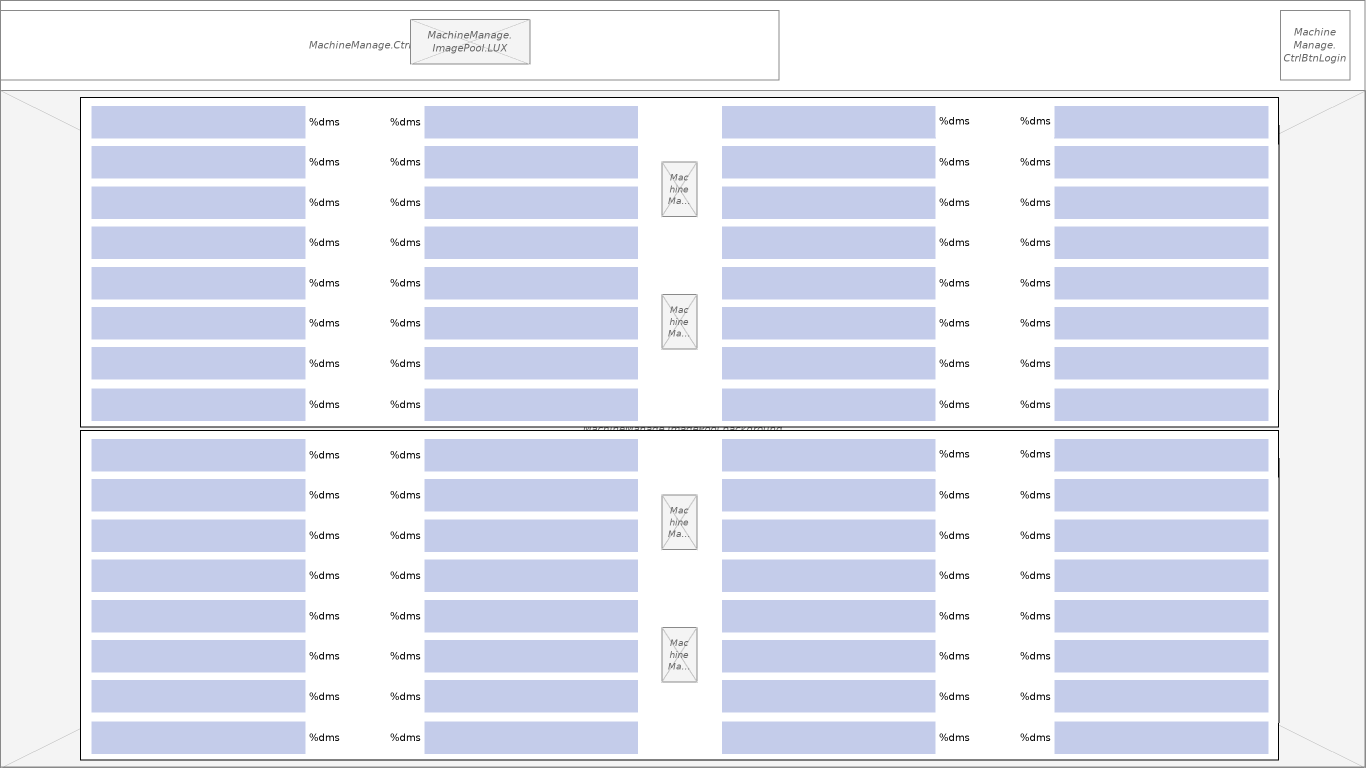
VISUALIZATION PageMonitor  // 1366x768
    Frame (0,0 1366x768)
        shows FrameMain()
    Frame (80,97 1200x330)
        shows CtrlInput(In := ADR(GVL_IO.I), SizeIn := Sizeof(GVL_IO.I), Enable := false, Ton := ADR(GVL_Data.stRecipe.arrInputTon), In_S := ADR(GVL.stShield_I))
    Frame (80,430 1200x330)
        shows CtrlOutput(In := ADR(GVL_IO.Q), SizeIn := sizeof(GVL_IO.Q), Enable := G_stSystem.stMode.bSetting, Ton := ADR(GVL_Data.stRecipe.arrOutputTon), In_S := ADR(GVL.stShield_Q))
END_VISUALIZATION

// ---- VISUs/PageSetting.TcVIS
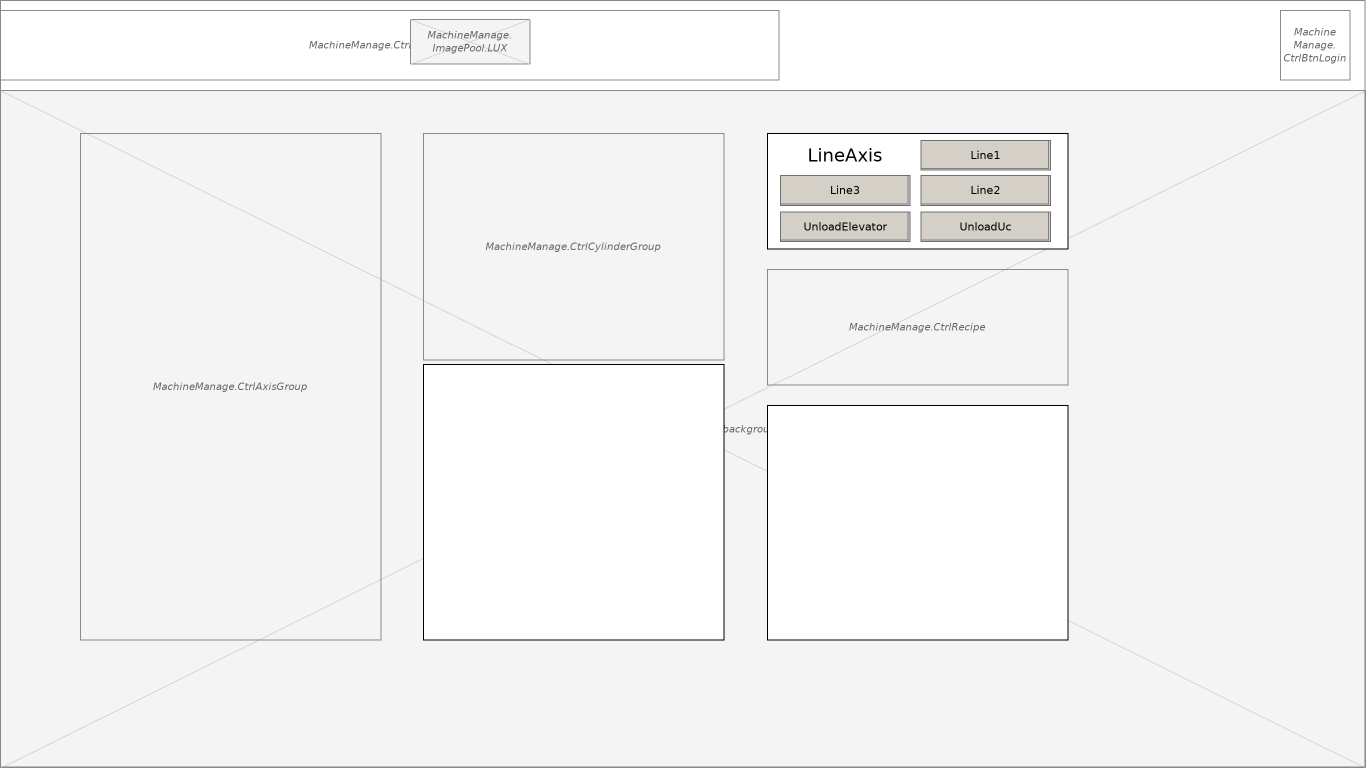
VISUALIZATION PageSetting  // 1366x768
    Frame (0,0 1366x768)
        shows FrameMain()
    Frame (80,133 301x507)
        shows MachineManage.CtrlAxisGroup(System := G_stSystem, Axis := G_arrAxis, Data := G_arrAxisData)
    Frame (423,133 301x227)
        shows MachineManage.CtrlCylinderGroup(System := G_stSystem, Cylinder := G_arrCylinder, CylinderData := G_arrCylinderData)
    RoundedRectangle (767,405 301x235), text list: 'ManualText', text index: 0
    Frame (767,269 301x116)
        shows MachineManage.CtrlRecipe()
    Frame (767,133 301x116)
        shows CtrlLine()
    RoundedRectangle (423,364 301x276), text list: 'ManualText', text index: 1
END_VISUALIZATION

